KUKA KRL program: fahrwege_big.src

&ACCESS RVO1
&REL 803
&COMMENT Rack 1 Place
&PARAM DISKPATH = KRC:\R1\Program\Unterprogramme
DEF  fahrwege_big( )
  ;FOLD INI;%{PE}
  ;FOLD BASISTECH INI
  GLOBAL INTERRUPT DECL 3 WHEN $STOPMESS==TRUE DO IR_STOPM ( )
  INTERRUPT ON 3
  BAS (#INITMOV,0 )
  ;ENDFOLD (BASISTECH INI)
  ;FOLD USER INI
  ;Make your modifications here

  ;ENDFOLD (USER INI)
  ;ENDFOLD (INI)

;***************************************************
; SAK herstellen
PTP $POS_ACT
;***************************************************

;---------------------------------
; Roboter in Grundstellung fahren
;---------------------------------
IF NOT ($IN_HOME OR $IN_HOME1 OR $IN_HOME2 OR $IN_HOME3) THEN
  UP_Rueckzug( )
ENDIF

;***************************************************
;      Unterprogramme fuer Produktionsbetrieb
;***************************************************

;***************************************************
; Satzanwahl auf gewuenschtes Unterprogramm
LOOP
  WAIT SEC 0.1
ENDLOOP
;***************************************************

HALT
UP_Place_R1_L1_S1( )
HALT
UP_Place_R1_L1_S2( )
HALT
UP_Place_R1_L1_S3( )
HALT
UP_Place_R1_L1_S4( )
HALT
UP_Place_R1_L2_S1( )
HALT
UP_Place_R1_L2_S2( )
HALT
UP_Place_R1_L2_S3( )
HALT
UP_Place_R1_L2_S4( )
HALT
UP_Place_R1_L3_S1( )
HALT
UP_Place_R1_L3_S2( )
HALT
UP_Place_R1_L3_S3( )
HALT
UP_Place_R1_L3_S4( )
HALT
UP_Place_R1_L4_S1( )
HALT
UP_Place_R1_L4_S2( )
HALT
UP_Place_R1_L4_S3( )
HALT
UP_Place_R1_L4_S4( )
HALT
UP_Place_R1_L5_S1( )
HALT
UP_Place_R1_L5_S2( )
HALT
UP_Place_R1_L5_S3( )
HALT
UP_Place_R1_L5_S4( )
HALT
UP_Place_R1_L6_S1( )
HALT
UP_Place_R1_L6_S2( )
HALT
UP_Place_R1_L6_S3( )
HALT
UP_Place_R1_L6_S4( )
HALT
UP_Place_R1_L7_S1( )
HALT
UP_Place_R1_L7_S2( )
HALT
UP_Place_R1_L7_S3( )
HALT
UP_Place_R1_L7_S4( )
HALT
UP_Place_R1_L8_S1( )
HALT
UP_Place_R1_L8_S2( )
HALT
UP_Place_R1_L8_S3( )
HALT
UP_Place_R1_L8_S4( )
HALT
UP_Rueckzug_R1Place( )
HALT
;***************************************************

END

; ##################################################

GLOBAL DEF UP_Place_R1_L1_S1( )
;***************************************************
; Place part on:
;    Rack  1
;    Level 1
;    Shelf 1
;***************************************************
;FOLD Preconditions - Vorraussetzungen
;***************************************************
; Enable collision detection
;FOLD COLLDETECT SetLimits Axis1: 150 % Axis2: 200 % Axis3: 150 % Axis4: 200 % Axis5: 150 % Axis6: 150 % ;%{PE}
;FOLD Parameters ;%{h}
;Params IlfProvider=kukaroboter.basistech.inlineforms.colldetect.setlimits; CollDetect.Command=SetLimits; CollDetect.Axis1=150; CollDetect.Axis2=200; CollDetect.Axis3=150; CollDetect.Axis4=200; CollDetect.Axis5=150; CollDetect.Axis6=150
;ENDFOLD
SET_TQ_VALUES(150, 200, 150, 200, 150, 150)
;ENDFOLD
;***************************************************
; Check for part in gripper (tool 2).
CheckPartPresent(OCCUPIED_GRIPPER,PART_ON_TOOL_2)
;***************************************************
; Enable part lost detection for tool 2
SetPartLostDetection(PART_ON_TOOL_2)
;***************************************************
; Set load data.
SetLoadData( )
;***************************************************
; Robot has to start from home position.
IF NOT $IN_HOME1 THEN
  UP_HomeToHome(1)
ENDIF
;***************************************************
;ENDFOLD

TRIGGER WHEN DISTANCE=1 DELAY=-1 DO Schrittmerker_R1Place(10002,10002,FHOME1,$nullframe,XHOME1) PRIO=-1
;FOLD PTP HOME1 Vel=12 % PHome1;%{PE}%R8.3.21,%MKUKATPBASIS,%CMOVE,%VPTP,%P 1:PTP, 2:HOME1, 3:, 5:12, 7:PHome1
$BWDSTART=FALSE
PDAT_ACT= PPHome1
FDAT_ACT= FHOME1
BAS(#PTP_PARAMS,12)
PTP XHOME1
;ENDFOLD

;***************************************************
;FOLD Area clearence handshake.
IF NOT $FLAG[M_Inbetriebnahme] THEN
  ;-------------------------------------------------
  ; Request area clearence.
  AnfStoer_Store1_1_A99=SET_REQUEST
  ;-------------------------------------------------
  ; Wait for area clearence from PLC.
  WAIT_FOR_INPUT("Frg_Storage1_1_E67",TRUE)
  ;-------------------------------------------------
  ; Reset area clearence request.
  AnfStoer_Store1_1_A99=RESET_REQUEST
  ;-------------------------------------------------
  ; start cyclic clearence check
  $CYCFLAG[ciFreigabeSPS]=Frg_Storage1_1_E67
  ;-------------------------------------------------
ENDIF
;***************************************************
; set "robot in area"
RobAusStorage1_1_A67=SET_IN_AREA
;ENDFOLD
;***************************************************

;***************************************************
;FOLD Check for Teachmode
IF $FLAG[M_Teachen] THEN
  WAIT FOR $T1
ENDIF
;ENDFOLD
;***************************************************

; move to the rack
TRIGGER WHEN DISTANCE=1 DELAY=-1 DO Schrittmerker_R1Place(10003,10002,FPlace_R1_L1_S1_VP1,XPlace_R1_L1_S1_VP1) PRIO=-1
;FOLD PTP Place_R1_L1_S1_VP1 CONT Vel=12 % PPlace_R1_L1_S1_VP1 Tool[2]:Lower Gripper Base[0];%{PE}%R8.3.21,%MKUKATPBASIS,%CMOVE,%VPTP,%P 1:PTP, 2:Place_R1_L1_S1_VP1, 3:C_DIS, 5:12, 7:PPlace_R1_L1_S1_VP1
$BWDSTART=FALSE
PDAT_ACT= PPPlace_R1_L1_S1_VP1
FDAT_ACT= FPlace_R1_L1_S1_VP1
BAS(#PTP_PARAMS,12)
PTP XPlace_R1_L1_S1_VP1 C_DIS
;ENDFOLD
TRIGGER WHEN DISTANCE=1 DELAY=-1 DO Schrittmerker_R1Place(10004,10003,FPlace_R1_L1_S1_VP2,XPlace_R1_L1_S1_VP2) PRIO=-1
;FOLD PTP Place_R1_L1_S1_VP2 CONT Vel=12 % PPlace_R1_L1_S1_VP2 Tool[2]:Lower Gripper Base[0];%{PE}%R8.3.21,%MKUKATPBASIS,%CMOVE,%VPTP,%P 1:PTP, 2:Place_R1_L1_S1_VP2, 3:C_DIS, 5:12, 7:PPlace_R1_L1_S1_VP2
$BWDSTART=FALSE
PDAT_ACT= PPPlace_R1_L1_S1_VP2
FDAT_ACT= FPlace_R1_L1_S1_VP2
BAS(#PTP_PARAMS,12)
PTP XPlace_R1_L1_S1_VP2 C_DIS
;ENDFOLD
TRIGGER WHEN DISTANCE=1 DELAY=-1 DO Schrittmerker_R1Place(10005,10004,FPlace_R1_L1_S1_VP3,XPlace_R1_L1_S1_VP3) PRIO=-1
;FOLD PTP Place_R1_L1_S1_VP3 CONT Vel=12 % PPlace_R1_L1_S1_VP3 Tool[2]:Lower Gripper Base[0];%{PE}%R8.3.21,%MKUKATPBASIS,%CMOVE,%VPTP,%P 1:PTP, 2:Place_R1_L1_S1_VP3, 3:C_DIS, 5:12, 7:PPlace_R1_L1_S1_VP3
$BWDSTART=FALSE
PDAT_ACT= PPPlace_R1_L1_S1_VP3
FDAT_ACT= FPlace_R1_L1_S1_VP3
BAS(#PTP_PARAMS,12)
PTP XPlace_R1_L1_S1_VP3 C_DIS
;ENDFOLD
TRIGGER WHEN DISTANCE=1 DELAY=-1 DO Schrittmerker_R1Place(10006,10005,FPlace_R1_L1_S1_VP4,XPlace_R1_L1_S1_VP4) PRIO=-1
;FOLD PTP Place_R1_L1_S1_VP4 CONT Vel=12 % PPlace_R1_L1_S1_VP4 Tool[2]:Lower Gripper Base[0];%{PE}%R8.3.21,%MKUKATPBASIS,%CMOVE,%VPTP,%P 1:PTP, 2:Place_R1_L1_S1_VP4, 3:C_DIS, 5:12, 7:PPlace_R1_L1_S1_VP4
$BWDSTART=FALSE
PDAT_ACT= PPPlace_R1_L1_S1_VP4
FDAT_ACT= FPlace_R1_L1_S1_VP4
BAS(#PTP_PARAMS,12)
PTP XPlace_R1_L1_S1_VP4 C_DIS
;ENDFOLD
TRIGGER WHEN DISTANCE=1 DELAY=-1 DO Schrittmerker_R1Place(10007,10006,FPlace_R1_L1_S1_VP5,XPlace_R1_L1_S1_VP5) PRIO=-1
;FOLD PTP Place_R1_L1_S1_VP5 CONT Vel=12 % PPlace_R1_L1_S1_VP5 Tool[2]:Lower Gripper Base[0];%{PE}%R8.3.21,%MKUKATPBASIS,%CMOVE,%VPTP,%P 1:PTP, 2:Place_R1_L1_S1_VP5, 3:C_DIS, 5:12, 7:PPlace_R1_L1_S1_VP5
$BWDSTART=FALSE
PDAT_ACT= PPPlace_R1_L1_S1_VP5
FDAT_ACT= FPlace_R1_L1_S1_VP5
BAS(#PTP_PARAMS,12)
PTP XPlace_R1_L1_S1_VP5 C_DIS
;ENDFOLD
TRIGGER WHEN DISTANCE=1 DELAY=-1 DO Schrittmerker_R1Place(10008,10007,FPlace_R1_L1_S1_VP6,XPlace_R1_L1_S1_VP6) PRIO=-1
;FOLD PTP Place_R1_L1_S1_VP6 CONT Vel=12 % PPlace_R1_L1_S1_VP6 Tool[2]:Lower Gripper Base[1]:Rack1;%{PE}%R8.3.21,%MKUKATPBASIS,%CMOVE,%VPTP,%P 1:PTP, 2:Place_R1_L1_S1_VP6, 3:C_DIS, 5:12, 7:PPlace_R1_L1_S1_VP6
$BWDSTART=FALSE
PDAT_ACT= PPPlace_R1_L1_S1_VP6
FDAT_ACT= FPlace_R1_L1_S1_VP6
BAS(#PTP_PARAMS,12)
PTP XPlace_R1_L1_S1_VP6 C_DIS
;ENDFOLD

TRIGGER WHEN DISTANCE=1 DELAY=-1 DO Schrittmerker_R1Place(10009,10008,FPlace_R1_L1_S1_Check,XPlace_R1_L1_S1_Check) PRIO=-1
;FOLD PTP Place_R1_L1_S1_Check Vel=12 % PPlace_R1_L1_S1_Check Tool[2]:Lower Gripper Base[1]:Rack1;%{PE}%R8.3.21,%MKUKATPBASIS,%CMOVE,%VPTP,%P 1:PTP, 2:Place_R1_L1_S1_Check, 3:, 5:12, 7:PPlace_R1_L1_S1_Check
$BWDSTART=FALSE
PDAT_ACT= PPPlace_R1_L1_S1_Check
FDAT_ACT= FPlace_R1_L1_S1_Check
BAS(#PTP_PARAMS,12)
PTP XPlace_R1_L1_S1_Check
;ENDFOLD

;***************************************************
;FOLD Pruefe Platz frei
IF (DetectPart(CHECK_SHELF,PLACE)==OCCUPIED) THEN
  UP_Rueckzug_R1Place( )
  RETURN
ENDIF
;ENDFOLD
;***************************************************

TRIGGER WHEN DISTANCE=1 DELAY=-1 DO Schrittmerker_R1Place(10010,10009,FPlace_R1_L1_S1_VP7,XPlace_R1_L1_S1_VP7) PRIO=-1
;FOLD LIN Place_R1_L1_S1_VP7 CONT Vel=0.5 m/s LPlace_R1_L1_S1_VP7 Tool[2]:Lower Gripper Base[1]:Rack1;%{PE}%R8.3.21,%MKUKATPBASIS,%CMOVE,%VLIN,%P 1:LIN, 2:Place_R1_L1_S1_VP7, 3:C_DIS C_DIS, 5:0.5, 7:LPlace_R1_L1_S1_VP7
$BWDSTART=FALSE
LDAT_ACT= LLPlace_R1_L1_S1_VP7
FDAT_ACT= FPlace_R1_L1_S1_VP7
BAS(#CP_PARAMS,0.5)
LIN XPlace_R1_L1_S1_VP7 C_DIS C_DIS
;ENDFOLD
TRIGGER WHEN DISTANCE=1 DELAY=-1 DO Schrittmerker_R1Place(10011,10010,FPlace_R1_L1_S1_VP8,XPlace_R1_L1_S1_VP8) PRIO=-1
;FOLD LIN Place_R1_L1_S1_VP8 CONT Vel=0.5 m/s LPlace_R1_L1_S1_VP8 Tool[2]:Lower Gripper Base[1]:Rack1;%{PE}%R8.3.21,%MKUKATPBASIS,%CMOVE,%VLIN,%P 1:LIN, 2:Place_R1_L1_S1_VP8, 3:C_DIS C_DIS, 5:0.5, 7:LPlace_R1_L1_S1_VP8
$BWDSTART=FALSE
LDAT_ACT= LLPlace_R1_L1_S1_VP8
FDAT_ACT= FPlace_R1_L1_S1_VP8
BAS(#CP_PARAMS,0.5)
LIN XPlace_R1_L1_S1_VP8 C_DIS C_DIS
;ENDFOLD
TRIGGER WHEN DISTANCE=1 DELAY=-1 DO Schrittmerker_R1Place(10012,10011,FPlace_R1_L1_S1_VP9,XPlace_R1_L1_S1_VP9) PRIO=-1
;FOLD LIN Place_R1_L1_S1_VP9 CONT Vel=0.5 m/s LPlace_R1_L1_S1_VP9 Tool[2]:Lower Gripper Base[1]:Rack1;%{PE}%R8.3.21,%MKUKATPBASIS,%CMOVE,%VLIN,%P 1:LIN, 2:Place_R1_L1_S1_VP9, 3:C_DIS C_DIS, 5:0.5, 7:LPlace_R1_L1_S1_VP9
$BWDSTART=FALSE
LDAT_ACT= LLPlace_R1_L1_S1_VP9
FDAT_ACT= FPlace_R1_L1_S1_VP9
BAS(#CP_PARAMS,0.5)
LIN XPlace_R1_L1_S1_VP9 C_DIS C_DIS
;ENDFOLD

;FOLD Test the way back home - part 1
CONTINUE
IF ($FLAG[M_Test_GrdstFahren1] AND NOT $FLAG[M_Test_GrdstFahren2]) THEN
  $FLAG[M_Test_GrdstFahren2]=TRUE
  UP_Rueckzug( )
  RETURN
ENDIF
;ENDFOLD

;-------------------------------
; Place part position
;-------------------------------
TRIGGER WHEN DISTANCE=1 DELAY=-1 DO Schrittmerker_R1Place(10013,10014,FPlace_R1_L1_S1_AP,XPlace_R1_L1_S1_AP) PRIO=-1
;FOLD LIN Place_R1_L1_S1_AP Vel=0.2 m/s LPlace_R1_L1_S1_AP Tool[2]:Lower Gripper Base[1]:Rack1;%{PE}%R8.3.21,%MKUKATPBASIS,%CMOVE,%VLIN,%P 1:LIN, 2:Place_R1_L1_S1_AP, 3:, 5:0.2, 7:LPlace_R1_L1_S1_AP
$BWDSTART=FALSE
LDAT_ACT= LLPlace_R1_L1_S1_AP
FDAT_ACT= FPlace_R1_L1_S1_AP
BAS(#CP_PARAMS,0.2)
LIN XPlace_R1_L1_S1_AP
;ENDFOLD

;FOLD Test the way back home - part 2
CONTINUE
IF $FLAG[M_Test_GrdstFahren2] THEN
  $FLAG[M_Test_GrdstFahren2]=FALSE
  UP_Rueckzug( )
  RETURN
ENDIF
;ENDFOLD

;***************************************************
; Disable part lost detection
SetPartLostDetection(NO_PART)
;***************************************************

TRIGGER WHEN DISTANCE=1 DELAY=-1 DO Schrittmerker_R1Place(10014,10015,FPlace_R1_L1_S1_NP1,XPlace_R1_L1_S1_NP1) PRIO=-1
;FOLD LIN Place_R1_L1_S1_NP1 Vel=0.2 m/s LPlace_R1_L1_S1_NP1 Tool[2]:Lower Gripper Base[1]:Rack 1 ;%{PE}
;FOLD Parameters ;%{h}
;Params IlfProvider=kukaroboter.basistech.inlineforms.movement.old; Kuka.IsGlobalPoint=False; Kuka.PointName=Place_R1_L1_S1_NP1; Kuka.BlendingEnabled=False; Kuka.MoveDataName=LPlace_R1_L1_S1_NP1; Kuka.VelocityPath=0.2; Kuka.CurrentCDSetIndex=0; Kuka.MovementParameterFieldEnabled=True; IlfCommand=LIN
;ENDFOLD
$BWDSTART = FALSE
LDAT_ACT = LLPlace_R1_L1_S1_NP1
FDAT_ACT = FPlace_R1_L1_S1_NP1
BAS(#CP_PARAMS, 0.2)
SET_CD_PARAMS (0)
LIN XPlace_R1_L1_S1_NP1
;ENDFOLD

;***************************************************
; Check for part present (empty gripper)
CheckPartPresent(EMPTY_GRIPPER)
;***************************************************
; set load data
SetLoadData( )
;***************************************************

TRIGGER WHEN DISTANCE=1 DELAY=-1 DO Schrittmerker_R1Place(10015,10016,FPlace_R1_L1_S1_NP2,XPlace_R1_L1_S1_NP2) PRIO=-1
;FOLD LIN Place_R1_L1_S1_NP2 CONT Vel=0.5 m/s LPlace_R1_L1_S1_NP2 Tool[2]:Lower Gripper Base[1]:Rack1;%{PE}%R8.3.21,%MKUKATPBASIS,%CMOVE,%VLIN,%P 1:LIN, 2:Place_R1_L1_S1_NP2, 3:C_DIS C_DIS, 5:0.5, 7:LPlace_R1_L1_S1_NP2
$BWDSTART=FALSE
LDAT_ACT= LLPlace_R1_L1_S1_NP2
FDAT_ACT= FPlace_R1_L1_S1_NP2
BAS(#CP_PARAMS,0.5)
LIN XPlace_R1_L1_S1_NP2 C_DIS C_DIS
;ENDFOLD
TRIGGER WHEN DISTANCE=1 DELAY=-1 DO Schrittmerker_R1Place(10016,10017,FPlace_R1_L1_S1_NP3,XPlace_R1_L1_S1_NP3) PRIO=-1
;FOLD LIN Place_R1_L1_S1_NP3 Vel=0.5 m/s LPlace_R1_L1_S1_NP3 Tool[2]:Lower Gripper Base[1]:Rack1;%{PE}%R8.3.21,%MKUKATPBASIS,%CMOVE,%VLIN,%P 1:LIN, 2:Place_R1_L1_S1_NP3, 3:, 5:0.5, 7:LPlace_R1_L1_S1_NP3
$BWDSTART=FALSE
LDAT_ACT= LLPlace_R1_L1_S1_NP3
FDAT_ACT= FPlace_R1_L1_S1_NP3
BAS(#CP_PARAMS,0.5)
LIN XPlace_R1_L1_S1_NP3
;ENDFOLD
TRIGGER WHEN DISTANCE=1 DELAY=-1 DO Schrittmerker_R1Place(10017,10018,FPlace_R1_L1_S1_NP4,XPlace_R1_L1_S1_NP4) PRIO=-1
;FOLD PTP Place_R1_L1_S1_NP4 CONT Vel=100 % PPlace_R1_L1_S1_NP4 Tool[2]:Lower Gripper Base[1]:Rack1;%{PE}%R8.3.21,%MKUKATPBASIS,%CMOVE,%VPTP,%P 1:PTP, 2:Place_R1_L1_S1_NP4, 3:C_DIS, 5:100, 7:PPlace_R1_L1_S1_NP4
$BWDSTART=FALSE
PDAT_ACT= PPPlace_R1_L1_S1_NP4
FDAT_ACT= FPlace_R1_L1_S1_NP4
BAS(#PTP_PARAMS,100)
PTP XPlace_R1_L1_S1_NP4 C_DIS
;ENDFOLD
TRIGGER WHEN DISTANCE=1 DELAY=-1 DO Schrittmerker_R1Place(10018,10019,FPlace_R1_L1_S1_NP5,XPlace_R1_L1_S1_NP5) PRIO=-1
;FOLD PTP Place_R1_L1_S1_NP5 CONT Vel=100 % PPlace_R1_L1_S1_NP5 Tool[2]:Lower Gripper Base[0];%{PE}%R8.3.21,%MKUKATPBASIS,%CMOVE,%VPTP,%P 1:PTP, 2:Place_R1_L1_S1_NP5, 3:C_DIS, 5:100, 7:PPlace_R1_L1_S1_NP5
$BWDSTART=FALSE
PDAT_ACT= PPPlace_R1_L1_S1_NP5
FDAT_ACT= FPlace_R1_L1_S1_NP5
BAS(#PTP_PARAMS,100)
PTP XPlace_R1_L1_S1_NP5 C_DIS
;ENDFOLD
TRIGGER WHEN DISTANCE=1 DELAY=-1 DO Schrittmerker_R1Place(10019,10020,FPlace_R1_L1_S1_NP6,XPlace_R1_L1_S1_NP6) PRIO=-1
;FOLD PTP Place_R1_L1_S1_NP6 CONT Vel=100 % PPlace_R1_L1_S1_NP6 Tool[2]:Lower Gripper Base[0];%{PE}%R8.3.21,%MKUKATPBASIS,%CMOVE,%VPTP,%P 1:PTP, 2:Place_R1_L1_S1_NP6, 3:C_DIS, 5:100, 7:PPlace_R1_L1_S1_NP6
$BWDSTART=FALSE
PDAT_ACT= PPPlace_R1_L1_S1_NP6
FDAT_ACT= FPlace_R1_L1_S1_NP6
BAS(#PTP_PARAMS,100)
PTP XPlace_R1_L1_S1_NP6 C_DIS
;ENDFOLD
TRIGGER WHEN DISTANCE=1 DELAY=-1 DO Schrittmerker_R1Place(10020,10021,FPlace_R1_L1_S1_NP7,XPlace_R1_L1_S1_NP7) PRIO=-1
;FOLD PTP Place_R1_L1_S1_NP7 CONT Vel=100 % PPlace_R1_L1_S1_NP7 Tool[2]:Lower Gripper Base[0];%{PE}%R8.3.21,%MKUKATPBASIS,%CMOVE,%VPTP,%P 1:PTP, 2:Place_R1_L1_S1_NP7, 3:C_DIS, 5:100, 7:PPlace_R1_L1_S1_NP7
$BWDSTART=FALSE
PDAT_ACT= PPPlace_R1_L1_S1_NP7
FDAT_ACT= FPlace_R1_L1_S1_NP7
BAS(#PTP_PARAMS,100)
PTP XPlace_R1_L1_S1_NP7 C_DIS
;ENDFOLD
TRIGGER WHEN DISTANCE=1 DELAY=-1 DO Schrittmerker_R1Place(10021,10022,FPlace_R1_L1_S1_NP8,XPlace_R1_L1_S1_NP8) PRIO=-1
;FOLD PTP Place_R1_L1_S1_NP8 CONT Vel=100 % PPlace_R1_L1_S1_NP8 Tool[2]:Lower Gripper Base[0];%{PE}%R8.3.21,%MKUKATPBASIS,%CMOVE,%VPTP,%P 1:PTP, 2:Place_R1_L1_S1_NP8, 3:C_DIS, 5:100, 7:PPlace_R1_L1_S1_NP8
$BWDSTART=FALSE
PDAT_ACT= PPPlace_R1_L1_S1_NP8
FDAT_ACT= FPlace_R1_L1_S1_NP8
BAS(#PTP_PARAMS,100)
PTP XPlace_R1_L1_S1_NP8 C_DIS
;ENDFOLD
TRIGGER WHEN DISTANCE=1 DELAY=-1 DO Schrittmerker_R1Place(10022,10023,FPlace_R1_L1_S1_NP9,XPlace_R1_L1_S1_NP9) PRIO=-1
;FOLD PTP Place_R1_L1_S1_NP9 CONT Vel=100 % PPlace_R1_L1_S1_NP9 Tool[2]:Lower Gripper Base[0];%{PE}%R8.3.21,%MKUKATPBASIS,%CMOVE,%VPTP,%P 1:PTP, 2:Place_R1_L1_S1_NP9, 3:C_DIS, 5:100, 7:PPlace_R1_L1_S1_NP9
$BWDSTART=FALSE
PDAT_ACT= PPPlace_R1_L1_S1_NP9
FDAT_ACT= FPlace_R1_L1_S1_NP9
BAS(#PTP_PARAMS,100)
PTP XPlace_R1_L1_S1_NP9 C_DIS
;ENDFOLD

TRIGGER WHEN DISTANCE=1 DELAY=-1 DO Schrittmerker_R1Place(10023,10002,FHOME1,$nullframe,XHOME1) PRIO=-1
;FOLD PTP HOME1 Vel=100 % PHome1;%{PE}%R8.3.21,%MKUKATPBASIS,%CMOVE,%VPTP,%P 1:PTP, 2:HOME1, 3:, 5:100, 7:PHome1
$BWDSTART=FALSE
PDAT_ACT= PPHome1
FDAT_ACT= FHOME1
BAS(#PTP_PARAMS,100)
PTP XHOME1
;ENDFOLD

;***************************************************
;FOLD Final tasks.
; Robot out of area Rack 1 Level 1
RobAusStorage1_1_A67=RESET_IN_AREA
;***************************************************
; stop cyclic clearence check
$CYCFLAG[ciFreigabeSPS]=DISABLE_MONITORING
;***************************************************
; Disable collision detection
;FOLD COLLDETECT Off ;%{PE}
;FOLD Parameters ;%{h}
;Params IlfProvider=kukaroboter.basistech.inlineforms.colldetect.off; CollDetect.Command=Off
;ENDFOLD
USE_CD_PARAMS(0)
;ENDFOLD
;***************************************************
;ENDFOLD
;***************************************************

END

; ##################################################

GLOBAL DEF UP_Place_R1_L1_S2( )
;***************************************************
; Place part on:
;    Rack  1
;    Level 1
;    Shelf 2
;***************************************************
;FOLD Preconditions - Vorraussetzungen
;***************************************************
; Enable collision detection
;FOLD COLLDETECT SetLimits Axis1: 150 % Axis2: 200 % Axis3: 150 % Axis4: 200 % Axis5: 150 % Axis6: 150 % ;%{PE}
;FOLD Parameters ;%{h}
;Params IlfProvider=kukaroboter.basistech.inlineforms.colldetect.setlimits; CollDetect.Command=SetLimits; CollDetect.Axis1=150; CollDetect.Axis2=200; CollDetect.Axis3=150; CollDetect.Axis4=200; CollDetect.Axis5=150; CollDetect.Axis6=150
;ENDFOLD
SET_TQ_VALUES(150, 200, 150, 200, 150, 150)
;ENDFOLD
;***************************************************
; Check for part in gripper (tool 2).
CheckPartPresent(OCCUPIED_GRIPPER,PART_ON_TOOL_2)
;***************************************************
; Enable part lost detection for tool 2
SetPartLostDetection(PART_ON_TOOL_2)
;***************************************************
; Set load data.
SetLoadData( )
;***************************************************
; Robot has to start from home position.
IF NOT $IN_HOME1 THEN
  UP_HomeToHome(1)
ENDIF
;***************************************************
;ENDFOLD

TRIGGER WHEN DISTANCE=1 DELAY=-1 DO Schrittmerker_R1Place(10002,10002,FHOME1,$nullframe,XHOME1) PRIO=-1
;FOLD PTP HOME1 Vel=12 % PHome1;%{PE}%R8.3.21,%MKUKATPBASIS,%CMOVE,%VPTP,%P 1:PTP, 2:HOME1, 3:, 5:12, 7:PHome1
$BWDSTART=FALSE
PDAT_ACT= PPHome1
FDAT_ACT= FHOME1
BAS(#PTP_PARAMS,12)
PTP XHOME1
;ENDFOLD

;***************************************************
;FOLD Area clearence handshake.
IF NOT $FLAG[M_Inbetriebnahme] THEN
  ;-------------------------------------------------
  ; Request area clearence.
  AnfStoer_Store1_1_A99=SET_REQUEST
  ;-------------------------------------------------
  ; Wait for area clearence from PLC.
  WAIT_FOR_INPUT("Frg_Storage1_1_E67",TRUE)
  ;-------------------------------------------------
  ; Reset area clearence request.
  AnfStoer_Store1_1_A99=RESET_REQUEST
  ;-------------------------------------------------
  ; start cyclic clearence check
  $CYCFLAG[ciFreigabeSPS]=Frg_Storage1_1_E67
  ;-------------------------------------------------
ENDIF
;***************************************************
; set "robot in area"
RobAusStorage1_1_A67=SET_IN_AREA
;ENDFOLD
;***************************************************

;***************************************************
;FOLD Check for Teachmode
IF $FLAG[M_Teachen] THEN
  WAIT FOR $T1
ENDIF
;ENDFOLD
;***************************************************

; move to the rack
TRIGGER WHEN DISTANCE=1 DELAY=-1 DO Schrittmerker_R1Place(10025,10002,FPlace_R1_L1_S2_VP1,XPlace_R1_L1_S2_VP1) PRIO=-1
;FOLD PTP Place_R1_L1_S2_VP1 CONT Vel=12 % PPlace_R1_L1_S2_VP1 Tool[2]:Lower Gripper Base[0];%{PE}%R8.3.21,%MKUKATPBASIS,%CMOVE,%VPTP,%P 1:PTP, 2:Place_R1_L1_S2_VP1, 3:C_DIS, 5:12, 7:PPlace_R1_L1_S2_VP1
$BWDSTART=FALSE
PDAT_ACT= PPPlace_R1_L1_S2_VP1
FDAT_ACT= FPlace_R1_L1_S2_VP1
BAS(#PTP_PARAMS,12)
PTP XPlace_R1_L1_S2_VP1 C_DIS
;ENDFOLD
TRIGGER WHEN DISTANCE=1 DELAY=-1 DO Schrittmerker_R1Place(10026,10025,FPlace_R1_L1_S2_VP2,XPlace_R1_L1_S2_VP2) PRIO=-1
;FOLD PTP Place_R1_L1_S2_VP2 CONT Vel=12 % PPlace_R1_L1_S2_VP2 Tool[2]:Lower Gripper Base[0];%{PE}%R8.3.21,%MKUKATPBASIS,%CMOVE,%VPTP,%P 1:PTP, 2:Place_R1_L1_S2_VP2, 3:C_DIS, 5:12, 7:PPlace_R1_L1_S2_VP2
$BWDSTART=FALSE
PDAT_ACT= PPPlace_R1_L1_S2_VP2
FDAT_ACT= FPlace_R1_L1_S2_VP2
BAS(#PTP_PARAMS,12)
PTP XPlace_R1_L1_S2_VP2 C_DIS
;ENDFOLD
TRIGGER WHEN DISTANCE=1 DELAY=-1 DO Schrittmerker_R1Place(10027,10026,FPlace_R1_L1_S2_VP3,XPlace_R1_L1_S2_VP3) PRIO=-1
;FOLD PTP Place_R1_L1_S2_VP3 CONT Vel=12 % PPlace_R1_L1_S2_VP3 Tool[2]:Lower Gripper Base[0];%{PE}%R8.3.21,%MKUKATPBASIS,%CMOVE,%VPTP,%P 1:PTP, 2:Place_R1_L1_S2_VP3, 3:C_DIS, 5:12, 7:PPlace_R1_L1_S2_VP3
$BWDSTART=FALSE
PDAT_ACT= PPPlace_R1_L1_S2_VP3
FDAT_ACT= FPlace_R1_L1_S2_VP3
BAS(#PTP_PARAMS,12)
PTP XPlace_R1_L1_S2_VP3 C_DIS
;ENDFOLD
TRIGGER WHEN DISTANCE=1 DELAY=-1 DO Schrittmerker_R1Place(10028,10027,FPlace_R1_L1_S2_VP4,XPlace_R1_L1_S2_VP4) PRIO=-1
;FOLD PTP Place_R1_L1_S2_VP4 CONT Vel=12 % PPlace_R1_L1_S2_VP4 Tool[2]:Lower Gripper Base[0];%{PE}%R8.3.21,%MKUKATPBASIS,%CMOVE,%VPTP,%P 1:PTP, 2:Place_R1_L1_S2_VP4, 3:C_DIS, 5:12, 7:PPlace_R1_L1_S2_VP4
$BWDSTART=FALSE
PDAT_ACT= PPPlace_R1_L1_S2_VP4
FDAT_ACT= FPlace_R1_L1_S2_VP4
BAS(#PTP_PARAMS,12)
PTP XPlace_R1_L1_S2_VP4 C_DIS
;ENDFOLD
TRIGGER WHEN DISTANCE=1 DELAY=-1 DO Schrittmerker_R1Place(10029,10028,FPlace_R1_L1_S2_VP5,XPlace_R1_L1_S2_VP5) PRIO=-1
;FOLD PTP Place_R1_L1_S2_VP5 CONT Vel=12 % PPlace_R1_L1_S2_VP5 Tool[2]:Lower Gripper Base[0];%{PE}%R8.3.21,%MKUKATPBASIS,%CMOVE,%VPTP,%P 1:PTP, 2:Place_R1_L1_S2_VP5, 3:C_DIS, 5:12, 7:PPlace_R1_L1_S2_VP5
$BWDSTART=FALSE
PDAT_ACT= PPPlace_R1_L1_S2_VP5
FDAT_ACT= FPlace_R1_L1_S2_VP5
BAS(#PTP_PARAMS,12)
PTP XPlace_R1_L1_S2_VP5 C_DIS
;ENDFOLD
TRIGGER WHEN DISTANCE=1 DELAY=-1 DO Schrittmerker_R1Place(10030,10029,FPlace_R1_L1_S2_VP6,XPlace_R1_L1_S2_VP6) PRIO=-1
;FOLD PTP Place_R1_L1_S2_VP6 CONT Vel=12 % PPlace_R1_L1_S2_VP6 Tool[2]:Lower Gripper Base[1]:Rack1;%{PE}%R8.3.21,%MKUKATPBASIS,%CMOVE,%VPTP,%P 1:PTP, 2:Place_R1_L1_S2_VP6, 3:C_DIS, 5:12, 7:PPlace_R1_L1_S2_VP6
$BWDSTART=FALSE
PDAT_ACT= PPPlace_R1_L1_S2_VP6
FDAT_ACT= FPlace_R1_L1_S2_VP6
BAS(#PTP_PARAMS,12)
PTP XPlace_R1_L1_S2_VP6 C_DIS
;ENDFOLD

TRIGGER WHEN DISTANCE=1 DELAY=-1 DO Schrittmerker_R1Place(10031,10030,FPlace_R1_L1_S2_Check,XPlace_R1_L1_S2_Check) PRIO=-1
;FOLD PTP Place_R1_L1_S2_Check Vel=12 % PPlace_R1_L1_S2_Check Tool[2]:Lower Gripper Base[1]:Rack1;%{PE}%R8.3.21,%MKUKATPBASIS,%CMOVE,%VPTP,%P 1:PTP, 2:Place_R1_L1_S2_Check, 3:, 5:12, 7:PPlace_R1_L1_S2_Check
$BWDSTART=FALSE
PDAT_ACT= PPPlace_R1_L1_S2_Check
FDAT_ACT= FPlace_R1_L1_S2_Check
BAS(#PTP_PARAMS,12)
PTP XPlace_R1_L1_S2_Check
;ENDFOLD

;***************************************************
;FOLD Pruefe Platz frei
IF (DetectPart(CHECK_SHELF,PLACE)==OCCUPIED) THEN
  UP_Rueckzug_R1Place( )
  RETURN
ENDIF
;ENDFOLD
;***************************************************

TRIGGER WHEN DISTANCE=1 DELAY=-1 DO Schrittmerker_R1Place(10032,10031,FPlace_R1_L1_S2_VP7,XPlace_R1_L1_S2_VP7) PRIO=-1
;FOLD LIN Place_R1_L1_S2_VP7 CONT Vel=0.5 m/s LPlace_R1_L1_S2_VP7 Tool[2]:Lower Gripper Base[1]:Rack1;%{PE}%R8.3.21,%MKUKATPBASIS,%CMOVE,%VLIN,%P 1:LIN, 2:Place_R1_L1_S2_VP7, 3:C_DIS C_DIS, 5:0.5, 7:LPlace_R1_L1_S2_VP7
$BWDSTART=FALSE
LDAT_ACT= LLPlace_R1_L1_S2_VP7
FDAT_ACT= FPlace_R1_L1_S2_VP7
BAS(#CP_PARAMS,0.5)
LIN XPlace_R1_L1_S2_VP7 C_DIS C_DIS
;ENDFOLD
TRIGGER WHEN DISTANCE=1 DELAY=-1 DO Schrittmerker_R1Place(10033,10032,FPlace_R1_L1_S2_VP8,XPlace_R1_L1_S2_VP8) PRIO=-1
;FOLD LIN Place_R1_L1_S2_VP8 CONT Vel=0.5 m/s LPlace_R1_L1_S2_VP8 Tool[2]:Lower Gripper Base[1]:Rack1;%{PE}%R8.3.21,%MKUKATPBASIS,%CMOVE,%VLIN,%P 1:LIN, 2:Place_R1_L1_S2_VP8, 3:C_DIS C_DIS, 5:0.5, 7:LPlace_R1_L1_S2_VP8
$BWDSTART=FALSE
LDAT_ACT= LLPlace_R1_L1_S2_VP8
FDAT_ACT= FPlace_R1_L1_S2_VP8
BAS(#CP_PARAMS,0.5)
LIN XPlace_R1_L1_S2_VP8 C_DIS C_DIS
;ENDFOLD

;FOLD Test the way back home - part 1
CONTINUE
IF ($FLAG[M_Test_GrdstFahren1] AND NOT $FLAG[M_Test_GrdstFahren2]) THEN
  $FLAG[M_Test_GrdstFahren2]=TRUE
  UP_Rueckzug( )
  RETURN
ENDIF
;ENDFOLD

;-------------------------------
; Place part position
;-------------------------------
TRIGGER WHEN DISTANCE=1 DELAY=-1 DO Schrittmerker_R1Place(10034,10035,FPlace_R1_L1_S2_AP,XPlace_R1_L1_S2_AP) PRIO=-1
;FOLD LIN Place_R1_L1_S2_AP Vel=0.2 m/s LPlace_R1_L1_S2_AP Tool[2]:Lower Gripper Base[1]:Rack1;%{PE}%R8.3.21,%MKUKATPBASIS,%CMOVE,%VLIN,%P 1:LIN, 2:Place_R1_L1_S2_AP, 3:, 5:0.2, 7:LPlace_R1_L1_S2_AP
$BWDSTART=FALSE
LDAT_ACT= LLPlace_R1_L1_S2_AP
FDAT_ACT= FPlace_R1_L1_S2_AP
BAS(#CP_PARAMS,0.2)
LIN XPlace_R1_L1_S2_AP
;ENDFOLD

;FOLD Test the way back home - part 2
CONTINUE
IF $FLAG[M_Test_GrdstFahren2] THEN
  $FLAG[M_Test_GrdstFahren2]=FALSE
  UP_Rueckzug( )
  RETURN
ENDIF
;ENDFOLD

;***************************************************
; Disable part lost detection
SetPartLostDetection(NO_PART)
;***************************************************

TRIGGER WHEN DISTANCE=1 DELAY=-1 DO Schrittmerker_R1Place(10035,10036,FPlace_R1_L1_S2_NP1,XPlace_R1_L1_S2_NP1) PRIO=-1
;FOLD LIN Place_R1_L1_S2_NP1 Vel=0.2 m/s LPlace_R1_L1_S2_NP1 Tool[2]:Lower Gripper Base[1]:Rack 1 ;%{PE}
;FOLD Parameters ;%{h}
;Params IlfProvider=kukaroboter.basistech.inlineforms.movement.old; Kuka.IsGlobalPoint=False; Kuka.PointName=Place_R1_L1_S2_NP1; Kuka.BlendingEnabled=True; Kuka.MoveDataName=LPlace_R1_L1_S2_NP1; Kuka.VelocityPath=0.2; Kuka.CurrentCDSetIndex=0; Kuka.MovementParameterFieldEnabled=True; IlfCommand=LIN
;ENDFOLD
$BWDSTART = FALSE
LDAT_ACT = LLPlace_R1_L1_S2_NP1
FDAT_ACT = FPlace_R1_L1_S2_NP1
BAS(#CP_PARAMS, 0.2)
SET_CD_PARAMS (0)
LIN XPlace_R1_L1_S2_NP1
;ENDFOLD

;***************************************************
; Check for part present (empty gripper)
CheckPartPresent(EMPTY_GRIPPER)
;***************************************************
; set load data
SetLoadData( )
;***************************************************

TRIGGER WHEN DISTANCE=1 DELAY=-1 DO Schrittmerker_R1Place(10036,10037,FPlace_R1_L1_S2_NP2,XPlace_R1_L1_S2_NP2) PRIO=-1
;FOLD LIN Place_R1_L1_S2_NP2 CONT Vel=0.5 m/s LPlace_R1_L1_S2_NP2 Tool[2]:Lower Gripper Base[1]:Rack1;%{PE}%R8.3.21,%MKUKATPBASIS,%CMOVE,%VLIN,%P 1:LIN, 2:Place_R1_L1_S2_NP2, 3:C_DIS C_DIS, 5:0.5, 7:LPlace_R1_L1_S2_NP2
$BWDSTART=FALSE
LDAT_ACT= LLPlace_R1_L1_S2_NP2
FDAT_ACT= FPlace_R1_L1_S2_NP2
BAS(#CP_PARAMS,0.5)
LIN XPlace_R1_L1_S2_NP2 C_DIS C_DIS
;ENDFOLD
TRIGGER WHEN DISTANCE=1 DELAY=-1 DO Schrittmerker_R1Place(10037,10038,FPlace_R1_L1_S2_NP3,XPlace_R1_L1_S2_NP3) PRIO=-1
;FOLD LIN Place_R1_L1_S2_NP3 CONT Vel=0.5 m/s LPlace_R1_L1_S2_NP3 Tool[2]:Lower Gripper Base[1]:Rack1;%{PE}%R8.3.21,%MKUKATPBASIS,%CMOVE,%VLIN,%P 1:LIN, 2:Place_R1_L1_S2_NP3, 3:C_DIS C_DIS, 5:0.5, 7:LPlace_R1_L1_S2_NP3
$BWDSTART=FALSE
LDAT_ACT= LLPlace_R1_L1_S2_NP3
FDAT_ACT= FPlace_R1_L1_S2_NP3
BAS(#CP_PARAMS,0.5)
LIN XPlace_R1_L1_S2_NP3 C_DIS C_DIS
;ENDFOLD
TRIGGER WHEN DISTANCE=1 DELAY=-1 DO Schrittmerker_R1Place(10038,10039,FPlace_R1_L1_S2_NP4,XPlace_R1_L1_S2_NP4) PRIO=-1
;FOLD PTP Place_R1_L1_S2_NP4 CONT Vel=100 % PPlace_R1_L1_S2_NP4 Tool[2]:Lower Gripper Base[0];%{PE}%R8.3.21,%MKUKATPBASIS,%CMOVE,%VPTP,%P 1:PTP, 2:Place_R1_L1_S2_NP4, 3:C_DIS, 5:100, 7:PPlace_R1_L1_S2_NP4
$BWDSTART=FALSE
PDAT_ACT= PPPlace_R1_L1_S2_NP4
FDAT_ACT= FPlace_R1_L1_S2_NP4
BAS(#PTP_PARAMS,100)
PTP XPlace_R1_L1_S2_NP4 C_DIS
;ENDFOLD
TRIGGER WHEN DISTANCE=1 DELAY=-1 DO Schrittmerker_R1Place(10039,10040,FPlace_R1_L1_S2_NP5,XPlace_R1_L1_S2_NP5) PRIO=-1
;FOLD PTP Place_R1_L1_S2_NP5 CONT Vel=100 % PPlace_R1_L1_S2_NP5 Tool[2]:Lower Gripper Base[0];%{PE}%R8.3.21,%MKUKATPBASIS,%CMOVE,%VPTP,%P 1:PTP, 2:Place_R1_L1_S2_NP5, 3:C_DIS, 5:100, 7:PPlace_R1_L1_S2_NP5
$BWDSTART=FALSE
PDAT_ACT= PPPlace_R1_L1_S2_NP5
FDAT_ACT= FPlace_R1_L1_S2_NP5
BAS(#PTP_PARAMS,100)
PTP XPlace_R1_L1_S2_NP5 C_DIS
;ENDFOLD
TRIGGER WHEN DISTANCE=1 DELAY=-1 DO Schrittmerker_R1Place(10040,10041,FPlace_R1_L1_S2_NP6,XPlace_R1_L1_S2_NP6) PRIO=-1
;FOLD PTP Place_R1_L1_S2_NP6 CONT Vel=100 % PPlace_R1_L1_S2_NP6 Tool[2]:Lower Gripper Base[0];%{PE}%R8.3.21,%MKUKATPBASIS,%CMOVE,%VPTP,%P 1:PTP, 2:Place_R1_L1_S2_NP6, 3:C_DIS, 5:100, 7:PPlace_R1_L1_S2_NP6
$BWDSTART=FALSE
PDAT_ACT= PPPlace_R1_L1_S2_NP6
FDAT_ACT= FPlace_R1_L1_S2_NP6
BAS(#PTP_PARAMS,100)
PTP XPlace_R1_L1_S2_NP6 C_DIS
;ENDFOLD
TRIGGER WHEN DISTANCE=1 DELAY=-1 DO Schrittmerker_R1Place(10041,10042,FPlace_R1_L1_S2_NP7,XPlace_R1_L1_S2_NP7) PRIO=-1
;FOLD PTP Place_R1_L1_S2_NP7 CONT Vel=100 % PPlace_R1_L1_S2_NP7 Tool[2]:Lower Gripper Base[0];%{PE}%R8.3.21,%MKUKATPBASIS,%CMOVE,%VPTP,%P 1:PTP, 2:Place_R1_L1_S2_NP7, 3:C_DIS, 5:100, 7:PPlace_R1_L1_S2_NP7
$BWDSTART=FALSE
PDAT_ACT= PPPlace_R1_L1_S2_NP7
FDAT_ACT= FPlace_R1_L1_S2_NP7
BAS(#PTP_PARAMS,100)
PTP XPlace_R1_L1_S2_NP7 C_DIS
;ENDFOLD
TRIGGER WHEN DISTANCE=1 DELAY=-1 DO Schrittmerker_R1Place(10042,10043,FPlace_R1_L1_S2_NP8,XPlace_R1_L1_S2_NP8) PRIO=-1
;FOLD PTP Place_R1_L1_S2_NP8 CONT Vel=100 % PPlace_R1_L1_S2_NP8 Tool[2]:Lower Gripper Base[0];%{PE}%R8.3.21,%MKUKATPBASIS,%CMOVE,%VPTP,%P 1:PTP, 2:Place_R1_L1_S2_NP8, 3:C_DIS, 5:100, 7:PPlace_R1_L1_S2_NP8
$BWDSTART=FALSE
PDAT_ACT= PPPlace_R1_L1_S2_NP8
FDAT_ACT= FPlace_R1_L1_S2_NP8
BAS(#PTP_PARAMS,100)
PTP XPlace_R1_L1_S2_NP8 C_DIS
;ENDFOLD

TRIGGER WHEN DISTANCE=1 DELAY=-1 DO Schrittmerker_R1Place(10043,10002,FHOME1,$nullframe,XHOME1) PRIO=-1
;FOLD PTP HOME1 Vel=100 % PHome1;%{PE}%R8.3.21,%MKUKATPBASIS,%CMOVE,%VPTP,%P 1:PTP, 2:HOME1, 3:, 5:100, 7:PHome1
$BWDSTART=FALSE
PDAT_ACT= PPHome1
FDAT_ACT= FHOME1
BAS(#PTP_PARAMS,100)
PTP XHOME1
;ENDFOLD

;***************************************************
;FOLD Final tasks.
; Robot out of area Rack 1 Level 1
RobAusStorage1_1_A67=RESET_IN_AREA
;***************************************************
; stop cyclic clearence check
$CYCFLAG[ciFreigabeSPS]=DISABLE_MONITORING
;***************************************************
; Disable collision detection
;FOLD COLLDETECT Off ;%{PE}
;FOLD Parameters ;%{h}
;Params IlfProvider=kukaroboter.basistech.inlineforms.colldetect.off; CollDetect.Command=Off
;ENDFOLD
USE_CD_PARAMS(0)
;ENDFOLD
;***************************************************
;ENDFOLD
;***************************************************

END

; ##################################################

GLOBAL DEF UP_Place_R1_L1_S3( )
;***************************************************
; Place part on:
;    Rack  1
;    Level 1
;    Shelf 3
;***************************************************
;FOLD Preconditions - Vorraussetzungen
;***************************************************
; Enable collision detection
;FOLD COLLDETECT SetLimits Axis1: 150 % Axis2: 200 % Axis3: 150 % Axis4: 200 % Axis5: 150 % Axis6: 150 % ;%{PE}
;FOLD Parameters ;%{h}
;Params IlfProvider=kukaroboter.basistech.inlineforms.colldetect.setlimits; CollDetect.Command=SetLimits; CollDetect.Axis1=150; CollDetect.Axis2=200; CollDetect.Axis3=150; CollDetect.Axis4=200; CollDetect.Axis5=150; CollDetect.Axis6=150
;ENDFOLD
SET_TQ_VALUES(150, 200, 150, 200, 150, 150)
;ENDFOLD
;***************************************************
; Check for part in gripper (tool 2).
CheckPartPresent(OCCUPIED_GRIPPER,PART_ON_TOOL_2)
;***************************************************
; Enable part lost detection for tool 2
SetPartLostDetection(PART_ON_TOOL_2)
;***************************************************
; Set load data.
SetLoadData( )
;***************************************************
; Robot has to start from home position.
IF NOT $IN_HOME1 THEN
  UP_HomeToHome(1)
ENDIF
;***************************************************
;ENDFOLD

TRIGGER WHEN DISTANCE=1 DELAY=-1 DO Schrittmerker_R1Place(10002,10002,FHOME1,$nullframe,XHOME1) PRIO=-1
;FOLD PTP HOME1 Vel=12 % PHome1;%{PE}%R8.3.21,%MKUKATPBASIS,%CMOVE,%VPTP,%P 1:PTP, 2:HOME1, 3:, 5:12, 7:PHome1
$BWDSTART=FALSE
PDAT_ACT= PPHome1
FDAT_ACT= FHOME1
BAS(#PTP_PARAMS,12)
PTP XHOME1
;ENDFOLD

;***************************************************
;FOLD Area clearence handshake.
IF NOT $FLAG[M_Inbetriebnahme] THEN
  ;-------------------------------------------------
  ; Request area clearence.
  AnfStoer_Store1_1_A99=SET_REQUEST
  ;-------------------------------------------------
  ; Wait for area clearence from PLC.
  WAIT_FOR_INPUT("Frg_Storage1_1_E67",TRUE)
  ;-------------------------------------------------
  ; Reset area clearence request.
  AnfStoer_Store1_1_A99=RESET_REQUEST
  ;-------------------------------------------------
  ; start cyclic clearence check
  $CYCFLAG[ciFreigabeSPS]=Frg_Storage1_1_E67
  ;-------------------------------------------------
ENDIF
;***************************************************
; set "robot in area"
RobAusStorage1_1_A67=SET_IN_AREA
;ENDFOLD
;***************************************************

;***************************************************
;FOLD Check for Teachmode
IF $FLAG[M_Teachen] THEN
  WAIT FOR $T1
ENDIF
;ENDFOLD
;***************************************************

; move to the rack
TRIGGER WHEN DISTANCE=1 DELAY=-1 DO Schrittmerker_R1Place(10045,10002,FPlace_R1_L1_S3_VP1,XPlace_R1_L1_S3_VP1) PRIO=-1
;FOLD PTP Place_R1_L1_S3_VP1 CONT Vel=12 % PPlace_R1_L1_S3_VP1 Tool[2]:Lower Gripper Base[0];%{PE}%R8.3.21,%MKUKATPBASIS,%CMOVE,%VPTP,%P 1:PTP, 2:Place_R1_L1_S3_VP1, 3:C_DIS, 5:12, 7:PPlace_R1_L1_S3_VP1
$BWDSTART=FALSE
PDAT_ACT= PPPlace_R1_L1_S3_VP1
FDAT_ACT= FPlace_R1_L1_S3_VP1
BAS(#PTP_PARAMS,12)
PTP XPlace_R1_L1_S3_VP1 C_DIS
;ENDFOLD
TRIGGER WHEN DISTANCE=1 DELAY=-1 DO Schrittmerker_R1Place(10046,10045,FPlace_R1_L1_S3_VP2,XPlace_R1_L1_S3_VP2) PRIO=-1
;FOLD PTP Place_R1_L1_S3_VP2 CONT Vel=12 % PPlace_R1_L1_S3_VP2 Tool[2]:Lower Gripper Base[0];%{PE}%R8.3.21,%MKUKATPBASIS,%CMOVE,%VPTP,%P 1:PTP, 2:Place_R1_L1_S3_VP2, 3:C_DIS, 5:12, 7:PPlace_R1_L1_S3_VP2
$BWDSTART=FALSE
PDAT_ACT= PPPlace_R1_L1_S3_VP2
FDAT_ACT= FPlace_R1_L1_S3_VP2
BAS(#PTP_PARAMS,12)
PTP XPlace_R1_L1_S3_VP2 C_DIS
;ENDFOLD
TRIGGER WHEN DISTANCE=1 DELAY=-1 DO Schrittmerker_R1Place(10047,10046,FPlace_R1_L1_S3_VP3,XPlace_R1_L1_S3_VP3) PRIO=-1
;FOLD PTP Place_R1_L1_S3_VP3 CONT Vel=12 % PPlace_R1_L1_S3_VP3 Tool[2]:Lower Gripper Base[0];%{PE}%R8.3.21,%MKUKATPBASIS,%CMOVE,%VPTP,%P 1:PTP, 2:Place_R1_L1_S3_VP3, 3:C_DIS, 5:12, 7:PPlace_R1_L1_S3_VP3
$BWDSTART=FALSE
PDAT_ACT= PPPlace_R1_L1_S3_VP3
FDAT_ACT= FPlace_R1_L1_S3_VP3
BAS(#PTP_PARAMS,12)
PTP XPlace_R1_L1_S3_VP3 C_DIS
;ENDFOLD
TRIGGER WHEN DISTANCE=1 DELAY=-1 DO Schrittmerker_R1Place(10048,10047,FPlace_R1_L1_S3_VP4,XPlace_R1_L1_S3_VP4) PRIO=-1
;FOLD PTP Place_R1_L1_S3_VP4 CONT Vel=12 % PPlace_R1_L1_S3_VP4 Tool[2]:Lower Gripper Base[0];%{PE}%R8.3.21,%MKUKATPBASIS,%CMOVE,%VPTP,%P 1:PTP, 2:Place_R1_L1_S3_VP4, 3:C_DIS, 5:12, 7:PPlace_R1_L1_S3_VP4
$BWDSTART=FALSE
PDAT_ACT= PPPlace_R1_L1_S3_VP4
FDAT_ACT= FPlace_R1_L1_S3_VP4
BAS(#PTP_PARAMS,12)
PTP XPlace_R1_L1_S3_VP4 C_DIS
;ENDFOLD
TRIGGER WHEN DISTANCE=1 DELAY=-1 DO Schrittmerker_R1Place(10049,10048,FPlace_R1_L1_S3_VP5,XPlace_R1_L1_S3_VP5) PRIO=-1
;FOLD PTP Place_R1_L1_S3_VP5 CONT Vel=12 % PPlace_R1_L1_S3_VP5 Tool[2]:Lower Gripper Base[0];%{PE}%R8.3.21,%MKUKATPBASIS,%CMOVE,%VPTP,%P 1:PTP, 2:Place_R1_L1_S3_VP5, 3:C_DIS, 5:12, 7:PPlace_R1_L1_S3_VP5
$BWDSTART=FALSE
PDAT_ACT= PPPlace_R1_L1_S3_VP5
FDAT_ACT= FPlace_R1_L1_S3_VP5
BAS(#PTP_PARAMS,12)
PTP XPlace_R1_L1_S3_VP5 C_DIS
;ENDFOLD
TRIGGER WHEN DISTANCE=1 DELAY=-1 DO Schrittmerker_R1Place(10050,10049,FPlace_R1_L1_S3_VP6,XPlace_R1_L1_S3_VP6) PRIO=-1
;FOLD PTP Place_R1_L1_S3_VP6 CONT Vel=12 % PPlace_R1_L1_S3_VP6 Tool[2]:Lower Gripper Base[1]:Rack1;%{PE}%R8.3.21,%MKUKATPBASIS,%CMOVE,%VPTP,%P 1:PTP, 2:Place_R1_L1_S3_VP6, 3:C_DIS, 5:12, 7:PPlace_R1_L1_S3_VP6
$BWDSTART=FALSE
PDAT_ACT= PPPlace_R1_L1_S3_VP6
FDAT_ACT= FPlace_R1_L1_S3_VP6
BAS(#PTP_PARAMS,12)
PTP XPlace_R1_L1_S3_VP6 C_DIS
;ENDFOLD

TRIGGER WHEN DISTANCE=1 DELAY=-1 DO Schrittmerker_R1Place(10051,10050,FPlace_R1_L1_S3_Check,XPlace_R1_L1_S3_Check) PRIO=-1
;FOLD PTP Place_R1_L1_S3_Check Vel=12 % PPlace_R1_L1_S3_Check Tool[2]:Lower Gripper Base[1]:Rack1;%{PE}%R8.3.21,%MKUKATPBASIS,%CMOVE,%VPTP,%P 1:PTP, 2:Place_R1_L1_S3_Check, 3:, 5:12, 7:PPlace_R1_L1_S3_Check
$BWDSTART=FALSE
PDAT_ACT= PPPlace_R1_L1_S3_Check
FDAT_ACT= FPlace_R1_L1_S3_Check
BAS(#PTP_PARAMS,12)
PTP XPlace_R1_L1_S3_Check
;ENDFOLD

;***************************************************
;FOLD Pruefe Platz frei
IF (DetectPart(CHECK_SHELF,PLACE)==OCCUPIED) THEN
  UP_Rueckzug_R1Place( )
  RETURN
ENDIF
;ENDFOLD
;***************************************************

TRIGGER WHEN DISTANCE=1 DELAY=-1 DO Schrittmerker_R1Place(10052,10051,FPlace_R1_L1_S3_VP7,XPlace_R1_L1_S3_VP7) PRIO=-1
;FOLD LIN Place_R1_L1_S3_VP7 CONT Vel=0.5 m/s LPlace_R1_L1_S3_VP7 Tool[2]:Lower Gripper Base[1]:Rack1;%{PE}%R8.3.21,%MKUKATPBASIS,%CMOVE,%VLIN,%P 1:LIN, 2:Place_R1_L1_S3_VP7, 3:C_DIS C_DIS, 5:0.5, 7:LPlace_R1_L1_S3_VP7
$BWDSTART=FALSE
LDAT_ACT= LLPlace_R1_L1_S3_VP7
FDAT_ACT= FPlace_R1_L1_S3_VP7
BAS(#CP_PARAMS,0.5)
LIN XPlace_R1_L1_S3_VP7 C_DIS C_DIS
;ENDFOLD
TRIGGER WHEN DISTANCE=1 DELAY=-1 DO Schrittmerker_R1Place(10053,10052,FPlace_R1_L1_S3_VP8,XPlace_R1_L1_S3_VP8) PRIO=-1
;FOLD LIN Place_R1_L1_S3_VP8 CONT Vel=0.5 m/s LPlace_R1_L1_S3_VP8 Tool[2]:Lower Gripper Base[1]:Rack1;%{PE}%R8.3.21,%MKUKATPBASIS,%CMOVE,%VLIN,%P 1:LIN, 2:Place_R1_L1_S3_VP8, 3:C_DIS C_DIS, 5:0.5, 7:LPlace_R1_L1_S3_VP8
$BWDSTART=FALSE
LDAT_ACT= LLPlace_R1_L1_S3_VP8
FDAT_ACT= FPlace_R1_L1_S3_VP8
BAS(#CP_PARAMS,0.5)
LIN XPlace_R1_L1_S3_VP8 C_DIS C_DIS
;ENDFOLD

;FOLD Test the way back home - part 1
CONTINUE
IF ($FLAG[M_Test_GrdstFahren1] AND NOT $FLAG[M_Test_GrdstFahren2]) THEN
  $FLAG[M_Test_GrdstFahren2]=TRUE
  UP_Rueckzug( )
  RETURN
ENDIF
;ENDFOLD

;-------------------------------
; Place part position
;-------------------------------
TRIGGER WHEN DISTANCE=1 DELAY=-1 DO Schrittmerker_R1Place(10054,10055,FPlace_R1_L1_S3_AP,XPlace_R1_L1_S3_AP) PRIO=-1
;FOLD LIN Place_R1_L1_S3_AP Vel=0.2 m/s LPlace_R1_L1_S3_AP Tool[2]:Lower Gripper Base[1]:Rack1;%{PE}%R8.3.21,%MKUKATPBASIS,%CMOVE,%VLIN,%P 1:LIN, 2:Place_R1_L1_S3_AP, 3:, 5:0.2, 7:LPlace_R1_L1_S3_AP
$BWDSTART=FALSE
LDAT_ACT= LLPlace_R1_L1_S3_AP
FDAT_ACT= FPlace_R1_L1_S3_AP
BAS(#CP_PARAMS,0.2)
LIN XPlace_R1_L1_S3_AP
;ENDFOLD

;FOLD Test the way back home - part 2
CONTINUE
IF $FLAG[M_Test_GrdstFahren2] THEN
  $FLAG[M_Test_GrdstFahren2]=FALSE
  UP_Rueckzug( )
  RETURN
ENDIF
;ENDFOLD

;***************************************************
; Disable part lost detection
SetPartLostDetection(NO_PART)
;***************************************************

TRIGGER WHEN DISTANCE=1 DELAY=-1 DO Schrittmerker_R1Place(10055,10056,FPlace_R1_L1_S3_NP1,XPlace_R1_L1_S3_NP1) PRIO=-1
;FOLD LIN Place_R1_L1_S3_NP1 Vel=0.2 m/s LPlace_R1_L1_S3_NP1 Tool[2]:Lower Gripper Base[1]:Rack1;%{PE}%R8.3.21,%MKUKATPBASIS,%CMOVE,%VLIN,%P 1:LIN, 2:Place_R1_L1_S3_NP1, 3:C_DIS C_DIS, 5:0.2, 7:LPlace_R1_L1_S3_NP1
$BWDSTART=FALSE
LDAT_ACT= LLPlace_R1_L1_S3_NP1
FDAT_ACT= FPlace_R1_L1_S3_NP1
BAS(#CP_PARAMS,0.2)
LIN XPlace_R1_L1_S3_NP1
;ENDFOLD

;***************************************************
; Check for part present (empty gripper)
CheckPartPresent(EMPTY_GRIPPER)
;***************************************************
; set load data
SetLoadData( )
;***************************************************

TRIGGER WHEN DISTANCE=1 DELAY=-1 DO Schrittmerker_R1Place(10056,10057,FPlace_R1_L1_S3_NP2,XPlace_R1_L1_S3_NP2) PRIO=-1
;FOLD LIN Place_R1_L1_S3_NP2 CONT Vel=0.5 m/s LPlace_R1_L1_S3_NP2 Tool[2]:Lower Gripper Base[1]:Rack1;%{PE}%R8.3.21,%MKUKATPBASIS,%CMOVE,%VLIN,%P 1:LIN, 2:Place_R1_L1_S3_NP2, 3:C_DIS C_DIS, 5:0.5, 7:LPlace_R1_L1_S3_NP2
$BWDSTART=FALSE
LDAT_ACT= LLPlace_R1_L1_S3_NP2
FDAT_ACT= FPlace_R1_L1_S3_NP2
BAS(#CP_PARAMS,0.5)
LIN XPlace_R1_L1_S3_NP2 C_DIS C_DIS
;ENDFOLD
TRIGGER WHEN DISTANCE=1 DELAY=-1 DO Schrittmerker_R1Place(10057,10058,FPlace_R1_L1_S3_NP3,XPlace_R1_L1_S3_NP3) PRIO=-1
;FOLD LIN Place_R1_L1_S3_NP3 CONT Vel=0.5 m/s LPlace_R1_L1_S3_NP3 Tool[2]:Lower Gripper Base[1]:Rack1;%{PE}%R8.3.21,%MKUKATPBASIS,%CMOVE,%VLIN,%P 1:LIN, 2:Place_R1_L1_S3_NP3, 3:C_DIS C_DIS, 5:0.5, 7:LPlace_R1_L1_S3_NP3
$BWDSTART=FALSE
LDAT_ACT= LLPlace_R1_L1_S3_NP3
FDAT_ACT= FPlace_R1_L1_S3_NP3
BAS(#CP_PARAMS,0.5)
LIN XPlace_R1_L1_S3_NP3 C_DIS C_DIS
;ENDFOLD
TRIGGER WHEN DISTANCE=1 DELAY=-1 DO Schrittmerker_R1Place(10058,10059,FPlace_R1_L1_S3_NP4,XPlace_R1_L1_S3_NP4) PRIO=-1
;FOLD PTP Place_R1_L1_S3_NP4 CONT Vel=100 % PPlace_R1_L1_S3_NP4 Tool[2]:Lower Gripper Base[0];%{PE}%R8.3.21,%MKUKATPBASIS,%CMOVE,%VPTP,%P 1:PTP, 2:Place_R1_L1_S3_NP4, 3:C_DIS, 5:100, 7:PPlace_R1_L1_S3_NP4
$BWDSTART=FALSE
PDAT_ACT= PPPlace_R1_L1_S3_NP4
FDAT_ACT= FPlace_R1_L1_S3_NP4
BAS(#PTP_PARAMS,100)
PTP XPlace_R1_L1_S3_NP4 C_DIS
;ENDFOLD
TRIGGER WHEN DISTANCE=1 DELAY=-1 DO Schrittmerker_R1Place(10059,10060,FPlace_R1_L1_S3_NP5,XPlace_R1_L1_S3_NP5) PRIO=-1
;FOLD PTP Place_R1_L1_S3_NP5 CONT Vel=100 % PPlace_R1_L1_S3_NP5 Tool[2]:Lower Gripper Base[0];%{PE}%R8.3.21,%MKUKATPBASIS,%CMOVE,%VPTP,%P 1:PTP, 2:Place_R1_L1_S3_NP5, 3:C_DIS, 5:100, 7:PPlace_R1_L1_S3_NP5
$BWDSTART=FALSE
PDAT_ACT= PPPlace_R1_L1_S3_NP5
FDAT_ACT= FPlace_R1_L1_S3_NP5
BAS(#PTP_PARAMS,100)
PTP XPlace_R1_L1_S3_NP5 C_DIS
;ENDFOLD
TRIGGER WHEN DISTANCE=1 DELAY=-1 DO Schrittmerker_R1Place(10060,10061,FPlace_R1_L1_S3_NP6,XPlace_R1_L1_S3_NP6) PRIO=-1
;FOLD PTP Place_R1_L1_S3_NP6 CONT Vel=100 % PPlace_R1_L1_S3_NP6 Tool[2]:Lower Gripper Base[0];%{PE}%R8.3.21,%MKUKATPBASIS,%CMOVE,%VPTP,%P 1:PTP, 2:Place_R1_L1_S3_NP6, 3:C_DIS, 5:100, 7:PPlace_R1_L1_S3_NP6
$BWDSTART=FALSE
PDAT_ACT= PPPlace_R1_L1_S3_NP6
FDAT_ACT= FPlace_R1_L1_S3_NP6
BAS(#PTP_PARAMS,100)
PTP XPlace_R1_L1_S3_NP6 C_DIS
;ENDFOLD
TRIGGER WHEN DISTANCE=1 DELAY=-1 DO Schrittmerker_R1Place(10061,10062,FPlace_R1_L1_S3_NP7,XPlace_R1_L1_S3_NP7) PRIO=-1
;FOLD PTP Place_R1_L1_S3_NP7 CONT Vel=100 % PPlace_R1_L1_S3_NP7 Tool[2]:Lower Gripper Base[0];%{PE}%R8.3.21,%MKUKATPBASIS,%CMOVE,%VPTP,%P 1:PTP, 2:Place_R1_L1_S3_NP7, 3:C_DIS, 5:100, 7:PPlace_R1_L1_S3_NP7
$BWDSTART=FALSE
PDAT_ACT= PPPlace_R1_L1_S3_NP7
FDAT_ACT= FPlace_R1_L1_S3_NP7
BAS(#PTP_PARAMS,100)
PTP XPlace_R1_L1_S3_NP7 C_DIS
;ENDFOLD
TRIGGER WHEN DISTANCE=1 DELAY=-1 DO Schrittmerker_R1Place(10062,10063,FPlace_R1_L1_S3_NP8,XPlace_R1_L1_S3_NP8) PRIO=-1
;FOLD PTP Place_R1_L1_S3_NP8 CONT Vel=100 % PPlace_R1_L1_S3_NP8 Tool[2]:Lower Gripper Base[0];%{PE}%R8.3.21,%MKUKATPBASIS,%CMOVE,%VPTP,%P 1:PTP, 2:Place_R1_L1_S3_NP8, 3:C_DIS, 5:100, 7:PPlace_R1_L1_S3_NP8
$BWDSTART=FALSE
PDAT_ACT= PPPlace_R1_L1_S3_NP8
FDAT_ACT= FPlace_R1_L1_S3_NP8
BAS(#PTP_PARAMS,100)
PTP XPlace_R1_L1_S3_NP8 C_DIS
;ENDFOLD

TRIGGER WHEN DISTANCE=1 DELAY=-1 DO Schrittmerker_R1Place(10063,10002,FHOME1,$nullframe,XHOME1) PRIO=-1
;FOLD PTP HOME1 Vel=100 % PHome1;%{PE}%R8.3.21,%MKUKATPBASIS,%CMOVE,%VPTP,%P 1:PTP, 2:HOME1, 3:, 5:100, 7:PHome1
$BWDSTART=FALSE
PDAT_ACT= PPHome1
FDAT_ACT= FHOME1
BAS(#PTP_PARAMS,100)
PTP XHOME1
;ENDFOLD

;***************************************************
;FOLD Final tasks.
; Robot out of area Rack 1 Level 1
RobAusStorage1_1_A67=RESET_IN_AREA
;***************************************************
; stop cyclic clearence check
$CYCFLAG[ciFreigabeSPS]=DISABLE_MONITORING
;***************************************************
; Disable collision detection
;FOLD COLLDETECT Off ;%{PE}
;FOLD Parameters ;%{h}
;Params IlfProvider=kukaroboter.basistech.inlineforms.colldetect.off; CollDetect.Command=Off
;ENDFOLD
USE_CD_PARAMS(0)
;ENDFOLD
;***************************************************
;ENDFOLD
;***************************************************

END

; ##################################################

GLOBAL DEF UP_Place_R1_L1_S4( )
;***************************************************
; Place part on:
;    Rack  1
;    Level 1
;    Shelf 4
;***************************************************
;FOLD Preconditions - Vorraussetzungen
;***************************************************
; Enable collision detection
;FOLD COLLDETECT SetLimits Axis1: 150 % Axis2: 200 % Axis3: 150 % Axis4: 200 % Axis5: 150 % Axis6: 150 % ;%{PE}
;FOLD Parameters ;%{h}
;Params IlfProvider=kukaroboter.basistech.inlineforms.colldetect.setlimits; CollDetect.Command=SetLimits; CollDetect.Axis1=150; CollDetect.Axis2=200; CollDetect.Axis3=150; CollDetect.Axis4=200; CollDetect.Axis5=150; CollDetect.Axis6=150
;ENDFOLD
SET_TQ_VALUES(150, 200, 150, 200, 150, 150)
;ENDFOLD
;***************************************************
; Check for part in gripper (tool 2).
CheckPartPresent(OCCUPIED_GRIPPER,PART_ON_TOOL_2)
;***************************************************
; Enable part lost detection for tool 2
SetPartLostDetection(PART_ON_TOOL_2)
;***************************************************
; Set load data.
SetLoadData( )
;***************************************************
; Robot has to start from home position.
IF NOT $IN_HOME1 THEN
  UP_HomeToHome(1)
ENDIF
;***************************************************
;ENDFOLD

TRIGGER WHEN DISTANCE=1 DELAY=-1 DO Schrittmerker_R1Place(10002,10002,FHOME1,$nullframe,XHOME1) PRIO=-1
;FOLD PTP HOME1 Vel=12 % PHome1;%{PE}%R8.3.21,%MKUKATPBASIS,%CMOVE,%VPTP,%P 1:PTP, 2:HOME1, 3:, 5:12, 7:PHome1
$BWDSTART=FALSE
PDAT_ACT= PPHome1
FDAT_ACT= FHOME1
BAS(#PTP_PARAMS,12)
PTP XHOME1
;ENDFOLD

;***************************************************
;FOLD Area clearence handshake.
IF NOT $FLAG[M_Inbetriebnahme] THEN
  ;-------------------------------------------------
  ; Request area clearence.
  AnfStoer_Store1_1_A99=SET_REQUEST
  ;-------------------------------------------------
  ; Wait for area clearence from PLC.
  WAIT_FOR_INPUT("Frg_Storage1_1_E67",TRUE)
  ;-------------------------------------------------
  ; Reset area clearence request.
  AnfStoer_Store1_1_A99=RESET_REQUEST
  ;-------------------------------------------------
  ; start cyclic clearence check
  $CYCFLAG[ciFreigabeSPS]=Frg_Storage1_1_E67
  ;-------------------------------------------------
ENDIF
;***************************************************
; set "robot in area"
RobAusStorage1_1_A67=SET_IN_AREA
;ENDFOLD
;***************************************************

;***************************************************
;FOLD Check for Teachmode
IF $FLAG[M_Teachen] THEN
  WAIT FOR $T1
ENDIF
;ENDFOLD
;***************************************************

; move to the rack
TRIGGER WHEN DISTANCE=1 DELAY=-1 DO Schrittmerker_R1Place(10065,10002,FPlace_R1_L1_S4_VP1,XPlace_R1_L1_S4_VP1) PRIO=-1
;FOLD PTP Place_R1_L1_S4_VP1 CONT Vel=12 % PPlace_R1_L1_S4_VP1 Tool[2]:Lower Gripper Base[0];%{PE}%R8.3.21,%MKUKATPBASIS,%CMOVE,%VPTP,%P 1:PTP, 2:Place_R1_L1_S4_VP1, 3:C_DIS, 5:12, 7:PPlace_R1_L1_S4_VP1
$BWDSTART=FALSE
PDAT_ACT= PPPlace_R1_L1_S4_VP1
FDAT_ACT= FPlace_R1_L1_S4_VP1
BAS(#PTP_PARAMS,12)
PTP XPlace_R1_L1_S4_VP1 C_DIS
;ENDFOLD
TRIGGER WHEN DISTANCE=1 DELAY=-1 DO Schrittmerker_R1Place(10066,10065,FPlace_R1_L1_S4_VP2,XPlace_R1_L1_S4_VP2) PRIO=-1
;FOLD PTP Place_R1_L1_S4_VP2 CONT Vel=12 % PPlace_R1_L1_S4_VP2 Tool[2]:Lower Gripper Base[0];%{PE}%R8.3.21,%MKUKATPBASIS,%CMOVE,%VPTP,%P 1:PTP, 2:Place_R1_L1_S4_VP2, 3:C_DIS, 5:12, 7:PPlace_R1_L1_S4_VP2
$BWDSTART=FALSE
PDAT_ACT= PPPlace_R1_L1_S4_VP2
FDAT_ACT= FPlace_R1_L1_S4_VP2
BAS(#PTP_PARAMS,12)
PTP XPlace_R1_L1_S4_VP2 C_DIS
;ENDFOLD
TRIGGER WHEN DISTANCE=1 DELAY=-1 DO Schrittmerker_R1Place(10067,10066,FPlace_R1_L1_S4_VP3,XPlace_R1_L1_S4_VP3) PRIO=-1
;FOLD PTP Place_R1_L1_S4_VP3 CONT Vel=12 % PPlace_R1_L1_S4_VP3 Tool[2]:Lower Gripper Base[0];%{PE}%R8.3.21,%MKUKATPBASIS,%CMOVE,%VPTP,%P 1:PTP, 2:Place_R1_L1_S4_VP3, 3:C_DIS, 5:12, 7:PPlace_R1_L1_S4_VP3
$BWDSTART=FALSE
PDAT_ACT= PPPlace_R1_L1_S4_VP3
FDAT_ACT= FPlace_R1_L1_S4_VP3
BAS(#PTP_PARAMS,12)
PTP XPlace_R1_L1_S4_VP3 C_DIS
;ENDFOLD
TRIGGER WHEN DISTANCE=1 DELAY=-1 DO Schrittmerker_R1Place(10068,10067,FPlace_R1_L1_S4_VP4,XPlace_R1_L1_S4_VP4) PRIO=-1
;FOLD PTP Place_R1_L1_S4_VP4 CONT Vel=12 % PPlace_R1_L1_S4_VP4 Tool[2]:Lower Gripper Base[0];%{PE}%R8.3.21,%MKUKATPBASIS,%CMOVE,%VPTP,%P 1:PTP, 2:Place_R1_L1_S4_VP4, 3:C_DIS, 5:12, 7:PPlace_R1_L1_S4_VP4
$BWDSTART=FALSE
PDAT_ACT= PPPlace_R1_L1_S4_VP4
FDAT_ACT= FPlace_R1_L1_S4_VP4
BAS(#PTP_PARAMS,12)
PTP XPlace_R1_L1_S4_VP4 C_DIS
;ENDFOLD
TRIGGER WHEN DISTANCE=1 DELAY=-1 DO Schrittmerker_R1Place(10069,10068,FPlace_R1_L1_S4_VP5,XPlace_R1_L1_S4_VP5) PRIO=-1
;FOLD PTP Place_R1_L1_S4_VP5 CONT Vel=12 % PPlace_R1_L1_S4_VP5 Tool[2]:Lower Gripper Base[0];%{PE}%R8.3.21,%MKUKATPBASIS,%CMOVE,%VPTP,%P 1:PTP, 2:Place_R1_L1_S4_VP5, 3:C_DIS, 5:12, 7:PPlace_R1_L1_S4_VP5
$BWDSTART=FALSE
PDAT_ACT= PPPlace_R1_L1_S4_VP5
FDAT_ACT= FPlace_R1_L1_S4_VP5
BAS(#PTP_PARAMS,12)
PTP XPlace_R1_L1_S4_VP5 C_DIS
;ENDFOLD
TRIGGER WHEN DISTANCE=1 DELAY=-1 DO Schrittmerker_R1Place(10070,10069,FPlace_R1_L1_S4_VP6,XPlace_R1_L1_S4_VP6) PRIO=-1
;FOLD PTP Place_R1_L1_S4_VP6 CONT Vel=12 % PPlace_R1_L1_S4_VP6 Tool[2]:Lower Gripper Base[1]:Rack1;%{PE}%R8.3.21,%MKUKATPBASIS,%CMOVE,%VPTP,%P 1:PTP, 2:Place_R1_L1_S4_VP6, 3:C_DIS, 5:12, 7:PPlace_R1_L1_S4_VP6
$BWDSTART=FALSE
PDAT_ACT= PPPlace_R1_L1_S4_VP6
FDAT_ACT= FPlace_R1_L1_S4_VP6
BAS(#PTP_PARAMS,12)
PTP XPlace_R1_L1_S4_VP6 C_DIS
;ENDFOLD

TRIGGER WHEN DISTANCE=1 DELAY=-1 DO Schrittmerker_R1Place(10071,10070,FPlace_R1_L1_S4_Check,XPlace_R1_L1_S4_Check) PRIO=-1
;FOLD PTP Place_R1_L1_S4_Check Vel=12 % PPlace_R1_L1_S4_Check Tool[2]:Lower Gripper Base[1]:Rack1;%{PE}%R8.3.21,%MKUKATPBASIS,%CMOVE,%VPTP,%P 1:PTP, 2:Place_R1_L1_S4_Check, 3:, 5:12, 7:PPlace_R1_L1_S4_Check
$BWDSTART=FALSE
PDAT_ACT= PPPlace_R1_L1_S4_Check
FDAT_ACT= FPlace_R1_L1_S4_Check
BAS(#PTP_PARAMS,12)
PTP XPlace_R1_L1_S4_Check
;ENDFOLD

;***************************************************
;FOLD Pruefe Platz frei
IF (DetectPart(CHECK_SHELF,PLACE)==OCCUPIED) THEN
  UP_Rueckzug_R1Place( )
  RETURN
ENDIF
;ENDFOLD
;***************************************************

TRIGGER WHEN DISTANCE=1 DELAY=-1 DO Schrittmerker_R1Place(10072,10071,FPlace_R1_L1_S4_VP7,XPlace_R1_L1_S4_VP7) PRIO=-1
;FOLD LIN Place_R1_L1_S4_VP7 CONT Vel=0.5 m/s LPlace_R1_L1_S4_VP7 Tool[2]:Lower Gripper Base[1]:Rack1;%{PE}%R8.3.21,%MKUKATPBASIS,%CMOVE,%VLIN,%P 1:LIN, 2:Place_R1_L1_S4_VP7, 3:C_DIS C_DIS, 5:0.5, 7:LPlace_R1_L1_S4_VP7
$BWDSTART=FALSE
LDAT_ACT= LLPlace_R1_L1_S4_VP7
FDAT_ACT= FPlace_R1_L1_S4_VP7
BAS(#CP_PARAMS,0.5)
LIN XPlace_R1_L1_S4_VP7 C_DIS C_DIS
;ENDFOLD
TRIGGER WHEN DISTANCE=1 DELAY=-1 DO Schrittmerker_R1Place(10073,10072,FPlace_R1_L1_S4_VP8,XPlace_R1_L1_S4_VP8) PRIO=-1
;FOLD LIN Place_R1_L1_S4_VP8 CONT Vel=0.5 m/s LPlace_R1_L1_S4_VP8 Tool[2]:Lower Gripper Base[1]:Rack1;%{PE}%R8.3.21,%MKUKATPBASIS,%CMOVE,%VLIN,%P 1:LIN, 2:Place_R1_L1_S4_VP8, 3:C_DIS C_DIS, 5:0.5, 7:LPlace_R1_L1_S4_VP8
$BWDSTART=FALSE
LDAT_ACT= LLPlace_R1_L1_S4_VP8
FDAT_ACT= FPlace_R1_L1_S4_VP8
BAS(#CP_PARAMS,0.5)
LIN XPlace_R1_L1_S4_VP8 C_DIS C_DIS
;ENDFOLD

;FOLD Test the way back home - part 1
CONTINUE
IF ($FLAG[M_Test_GrdstFahren1] AND NOT $FLAG[M_Test_GrdstFahren2]) THEN
  $FLAG[M_Test_GrdstFahren2]=TRUE
  UP_Rueckzug( )
  RETURN
ENDIF
;ENDFOLD

;-------------------------------
; Place part position
;-------------------------------
TRIGGER WHEN DISTANCE=1 DELAY=-1 DO Schrittmerker_R1Place(10074,10075,FPlace_R1_L1_S4_AP,XPlace_R1_L1_S4_AP) PRIO=-1
;FOLD LIN Place_R1_L1_S4_AP Vel=0.2 m/s LPlace_R1_L1_S4_AP Tool[2]:Lower Gripper Base[1]:Rack1;%{PE}%R8.3.21,%MKUKATPBASIS,%CMOVE,%VLIN,%P 1:LIN, 2:Place_R1_L1_S4_AP, 3:, 5:0.2, 7:LPlace_R1_L1_S4_AP
$BWDSTART=FALSE
LDAT_ACT= LLPlace_R1_L1_S4_AP
FDAT_ACT= FPlace_R1_L1_S4_AP
BAS(#CP_PARAMS,0.2)
LIN XPlace_R1_L1_S4_AP
;ENDFOLD

;FOLD Test the way back home - part 2
CONTINUE
IF $FLAG[M_Test_GrdstFahren2] THEN
  $FLAG[M_Test_GrdstFahren2]=FALSE
  UP_Rueckzug( )
  RETURN
ENDIF
;ENDFOLD

;***************************************************
; Disable part lost detection
SetPartLostDetection(NO_PART)
;***************************************************

TRIGGER WHEN DISTANCE=1 DELAY=-1 DO Schrittmerker_R1Place(10075,10076,FPlace_R1_L1_S4_NP1,XPlace_R1_L1_S4_NP1) PRIO=-1
;FOLD LIN Place_R1_L1_S4_NP1 Vel=0.2 m/s LPlace_R1_L1_S4_NP1 Tool[2]:Lower Gripper Base[1]:Rack 1 ;%{PE}
;FOLD Parameters ;%{h}
;Params IlfProvider=kukaroboter.basistech.inlineforms.movement.old; Kuka.IsGlobalPoint=False; Kuka.PointName=Place_R1_L1_S4_NP1; Kuka.BlendingEnabled=False; Kuka.MoveDataName=LPlace_R1_L1_S4_NP1; Kuka.VelocityPath=0.2; Kuka.CurrentCDSetIndex=0; Kuka.MovementParameterFieldEnabled=True; IlfCommand=LIN
;ENDFOLD
$BWDSTART = FALSE
LDAT_ACT = LLPlace_R1_L1_S4_NP1
FDAT_ACT = FPlace_R1_L1_S4_NP1
BAS(#CP_PARAMS, 0.2)
SET_CD_PARAMS (0)
LIN XPlace_R1_L1_S4_NP1
;ENDFOLD

;***************************************************
; Check for part present (empty gripper)
CheckPartPresent(EMPTY_GRIPPER)
;***************************************************
; set load data
SetLoadData( )
;***************************************************

TRIGGER WHEN DISTANCE=1 DELAY=-1 DO Schrittmerker_R1Place(10076,10077,FPlace_R1_L1_S4_NP2,XPlace_R1_L1_S4_NP2) PRIO=-1
;FOLD LIN Place_R1_L1_S4_NP2 CONT Vel=0.5 m/s LPlace_R1_L1_S4_NP2 Tool[2]:Lower Gripper Base[1]:Rack1;%{PE}%R8.3.21,%MKUKATPBASIS,%CMOVE,%VLIN,%P 1:LIN, 2:Place_R1_L1_S4_NP2, 3:C_DIS C_DIS, 5:0.5, 7:LPlace_R1_L1_S4_NP2
$BWDSTART=FALSE
LDAT_ACT= LLPlace_R1_L1_S4_NP2
FDAT_ACT= FPlace_R1_L1_S4_NP2
BAS(#CP_PARAMS,0.5)
LIN XPlace_R1_L1_S4_NP2 C_DIS C_DIS
;ENDFOLD
TRIGGER WHEN DISTANCE=1 DELAY=-1 DO Schrittmerker_R1Place(10077,10078,FPlace_R1_L1_S4_NP3,XPlace_R1_L1_S4_NP3) PRIO=-1
;FOLD LIN Place_R1_L1_S4_NP3 CONT Vel=0.5 m/s LPlace_R1_L1_S4_NP3 Tool[2]:Lower Gripper Base[1]:Rack1;%{PE}%R8.3.21,%MKUKATPBASIS,%CMOVE,%VLIN,%P 1:LIN, 2:Place_R1_L1_S4_NP3, 3:C_DIS C_DIS, 5:0.5, 7:LPlace_R1_L1_S4_NP3
$BWDSTART=FALSE
LDAT_ACT= LLPlace_R1_L1_S4_NP3
FDAT_ACT= FPlace_R1_L1_S4_NP3
BAS(#CP_PARAMS,0.5)
LIN XPlace_R1_L1_S4_NP3 C_DIS C_DIS
;ENDFOLD
TRIGGER WHEN DISTANCE=1 DELAY=-1 DO Schrittmerker_R1Place(10078,10079,FPlace_R1_L1_S4_NP4,XPlace_R1_L1_S4_NP4) PRIO=-1
;FOLD PTP Place_R1_L1_S4_NP4 CONT Vel=100 % PPlace_R1_L1_S4_NP4 Tool[2]:Lower Gripper Base[0];%{PE}%R8.3.21,%MKUKATPBASIS,%CMOVE,%VPTP,%P 1:PTP, 2:Place_R1_L1_S4_NP4, 3:C_DIS, 5:100, 7:PPlace_R1_L1_S4_NP4
$BWDSTART=FALSE
PDAT_ACT= PPPlace_R1_L1_S4_NP4
FDAT_ACT= FPlace_R1_L1_S4_NP4
BAS(#PTP_PARAMS,100)
PTP XPlace_R1_L1_S4_NP4 C_DIS
;ENDFOLD
TRIGGER WHEN DISTANCE=1 DELAY=-1 DO Schrittmerker_R1Place(10079,10080,FPlace_R1_L1_S4_NP5,XPlace_R1_L1_S4_NP5) PRIO=-1
;FOLD PTP Place_R1_L1_S4_NP5 CONT Vel=100 % PPlace_R1_L1_S4_NP5 Tool[2]:Lower Gripper Base[0];%{PE}%R8.3.21,%MKUKATPBASIS,%CMOVE,%VPTP,%P 1:PTP, 2:Place_R1_L1_S4_NP5, 3:C_DIS, 5:100, 7:PPlace_R1_L1_S4_NP5
$BWDSTART=FALSE
PDAT_ACT= PPPlace_R1_L1_S4_NP5
FDAT_ACT= FPlace_R1_L1_S4_NP5
BAS(#PTP_PARAMS,100)
PTP XPlace_R1_L1_S4_NP5 C_DIS
;ENDFOLD
TRIGGER WHEN DISTANCE=1 DELAY=-1 DO Schrittmerker_R1Place(10080,10081,FPlace_R1_L1_S4_NP6,XPlace_R1_L1_S4_NP6) PRIO=-1
;FOLD PTP Place_R1_L1_S4_NP6 CONT Vel=100 % PPlace_R1_L1_S4_NP6 Tool[2]:Lower Gripper Base[0];%{PE}%R8.3.21,%MKUKATPBASIS,%CMOVE,%VPTP,%P 1:PTP, 2:Place_R1_L1_S4_NP6, 3:C_DIS, 5:100, 7:PPlace_R1_L1_S4_NP6
$BWDSTART=FALSE
PDAT_ACT= PPPlace_R1_L1_S4_NP6
FDAT_ACT= FPlace_R1_L1_S4_NP6
BAS(#PTP_PARAMS,100)
PTP XPlace_R1_L1_S4_NP6 C_DIS
;ENDFOLD
TRIGGER WHEN DISTANCE=1 DELAY=-1 DO Schrittmerker_R1Place(10081,10082,FPlace_R1_L1_S4_NP7,XPlace_R1_L1_S4_NP7) PRIO=-1
;FOLD PTP Place_R1_L1_S4_NP7 CONT Vel=100 % PPlace_R1_L1_S4_NP7 Tool[2]:Lower Gripper Base[0];%{PE}%R8.3.21,%MKUKATPBASIS,%CMOVE,%VPTP,%P 1:PTP, 2:Place_R1_L1_S4_NP7, 3:C_DIS, 5:100, 7:PPlace_R1_L1_S4_NP7
$BWDSTART=FALSE
PDAT_ACT= PPPlace_R1_L1_S4_NP7
FDAT_ACT= FPlace_R1_L1_S4_NP7
BAS(#PTP_PARAMS,100)
PTP XPlace_R1_L1_S4_NP7 C_DIS
;ENDFOLD
TRIGGER WHEN DISTANCE=1 DELAY=-1 DO Schrittmerker_R1Place(10082,10083,FPlace_R1_L1_S4_NP8,XPlace_R1_L1_S4_NP8) PRIO=-1
;FOLD PTP Place_R1_L1_S4_NP8 CONT Vel=100 % PPlace_R1_L1_S4_NP8 Tool[2]:Lower Gripper Base[0];%{PE}%R8.3.21,%MKUKATPBASIS,%CMOVE,%VPTP,%P 1:PTP, 2:Place_R1_L1_S4_NP8, 3:C_DIS, 5:100, 7:PPlace_R1_L1_S4_NP8
$BWDSTART=FALSE
PDAT_ACT= PPPlace_R1_L1_S4_NP8
FDAT_ACT= FPlace_R1_L1_S4_NP8
BAS(#PTP_PARAMS,100)
PTP XPlace_R1_L1_S4_NP8 C_DIS
;ENDFOLD

TRIGGER WHEN DISTANCE=1 DELAY=-1 DO Schrittmerker_R1Place(10083,10002,FHOME1,$nullframe,XHOME1) PRIO=-1
;FOLD PTP HOME1 Vel=100 % PHome1;%{PE}%R8.3.21,%MKUKATPBASIS,%CMOVE,%VPTP,%P 1:PTP, 2:HOME1, 3:, 5:100, 7:PHome1
$BWDSTART=FALSE
PDAT_ACT= PPHome1
FDAT_ACT= FHOME1
BAS(#PTP_PARAMS,100)
PTP XHOME1
;ENDFOLD

;***************************************************
;FOLD Final tasks.
; Robot out of area Rack 1 Level 1
RobAusStorage1_1_A67=RESET_IN_AREA
;***************************************************
; stop cyclic clearence check
$CYCFLAG[ciFreigabeSPS]=DISABLE_MONITORING
;***************************************************
; Disable collision detection
;FOLD COLLDETECT Off ;%{PE}
;FOLD Parameters ;%{h}
;Params IlfProvider=kukaroboter.basistech.inlineforms.colldetect.off; CollDetect.Command=Off
;ENDFOLD
USE_CD_PARAMS(0)
;ENDFOLD
;***************************************************
;ENDFOLD
;***************************************************

END

; ##################################################

GLOBAL DEF UP_Place_R1_L2_S1( )
;***************************************************
; Place part on:
;    Rack  1
;    Level 2
;    Shelf 1
;  RBG Kollision beachten!
;***************************************************
;FOLD Preconditions - Vorraussetzungen
;***************************************************
; Enable collision detection
;FOLD COLLDETECT SetLimits Axis1: 150 % Axis2: 200 % Axis3: 150 % Axis4: 200 % Axis5: 150 % Axis6: 150 % ;%{PE}
;FOLD Parameters ;%{h}
;Params IlfProvider=kukaroboter.basistech.inlineforms.colldetect.setlimits; CollDetect.Command=SetLimits; CollDetect.Axis1=150; CollDetect.Axis2=200; CollDetect.Axis3=150; CollDetect.Axis4=200; CollDetect.Axis5=150; CollDetect.Axis6=150
;ENDFOLD
SET_TQ_VALUES(150, 200, 150, 200, 150, 150)
;ENDFOLD
;***************************************************
; Check for part in gripper (tool 2).
CheckPartPresent(OCCUPIED_GRIPPER,PART_ON_TOOL_2)
;***************************************************
; Enable part lost detection for tool 2
SetPartLostDetection(PART_ON_TOOL_2)
;***************************************************
; Set load data.
SetLoadData( )
;***************************************************
; Robot has to start from home position.
IF NOT $IN_HOME1 THEN
  UP_HomeToHome(1)
ENDIF
;***************************************************
;ENDFOLD

TRIGGER WHEN DISTANCE=1 DELAY=-1 DO Schrittmerker_R1Place(10002,10002,FHOME1,$nullframe,XHOME1) PRIO=-1
;FOLD PTP HOME1 Vel=12 % PHome1;%{PE}%R8.3.21,%MKUKATPBASIS,%CMOVE,%VPTP,%P 1:PTP, 2:HOME1, 3:, 5:12, 7:PHome1
$BWDSTART=FALSE
PDAT_ACT= PPHome1
FDAT_ACT= FHOME1
BAS(#PTP_PARAMS,12)
PTP XHOME1
;ENDFOLD

;***************************************************
;FOLD Area clearence handshake.
IF NOT $FLAG[M_Inbetriebnahme] THEN
  ;-------------------------------------------------
  ; Request area clearence.
  AnfStoer_Store1_2_A100=SET_REQUEST
  ;-------------------------------------------------
  ; Wait for area clearence from PLC.
  WAIT_FOR_INPUT("Frg_Storage1_2_E68",TRUE)
  ;-------------------------------------------------
  ; Reset area clearence request.
  AnfStoer_Store1_2_A100=RESET_REQUEST
  ;-------------------------------------------------
  ; start cyclic clearence check
  $CYCFLAG[ciFreigabeSPS]=Frg_Storage1_2_E68
  ;-------------------------------------------------
ENDIF
;***************************************************
; set "robot in area"
RobAusStorage1_2_A68=SET_IN_AREA
;ENDFOLD
;***************************************************

;***************************************************
;FOLD Check for Teachmode
IF $FLAG[M_Teachen] THEN
  WAIT FOR $T1
ENDIF
;ENDFOLD
;***************************************************

; move to the rack
TRIGGER WHEN DISTANCE=1 DELAY=-1 DO Schrittmerker_R1Place(10085,10002,FPlace_R1_L2_S1_VP1,XPlace_R1_L2_S1_VP1) PRIO=-1
;FOLD PTP Place_R1_L2_S1_VP1 CONT Vel=12 % PPlace_R1_L2_S1_VP1 Tool[2]:Lower Gripper Base[0];%{PE}%R8.3.21,%MKUKATPBASIS,%CMOVE,%VPTP,%P 1:PTP, 2:Place_R1_L2_S1_VP1, 3:C_DIS, 5:12, 7:PPlace_R1_L2_S1_VP1
$BWDSTART=FALSE
PDAT_ACT= PPPlace_R1_L2_S1_VP1
FDAT_ACT= FPlace_R1_L2_S1_VP1
BAS(#PTP_PARAMS,12)
PTP XPlace_R1_L2_S1_VP1 C_DIS
;ENDFOLD
TRIGGER WHEN DISTANCE=1 DELAY=-1 DO Schrittmerker_R1Place(10086,10085,FPlace_R1_L2_S1_VP2,XPlace_R1_L2_S1_VP2) PRIO=-1
;FOLD PTP Place_R1_L2_S1_VP2 CONT Vel=12 % PPlace_R1_L2_S1_VP2 Tool[2]:Lower Gripper Base[0];%{PE}%R8.3.21,%MKUKATPBASIS,%CMOVE,%VPTP,%P 1:PTP, 2:Place_R1_L2_S1_VP2, 3:C_DIS, 5:12, 7:PPlace_R1_L2_S1_VP2
$BWDSTART=FALSE
PDAT_ACT= PPPlace_R1_L2_S1_VP2
FDAT_ACT= FPlace_R1_L2_S1_VP2
BAS(#PTP_PARAMS,12)
PTP XPlace_R1_L2_S1_VP2 C_DIS
;ENDFOLD
TRIGGER WHEN DISTANCE=1 DELAY=-1 DO Schrittmerker_R1Place(10087,10086,FPlace_R1_L2_S1_VP3,XPlace_R1_L2_S1_VP3) PRIO=-1
;FOLD PTP Place_R1_L2_S1_VP3 CONT Vel=12 % PPlace_R1_L2_S1_VP3 Tool[2]:Lower Gripper Base[0];%{PE}%R8.3.21,%MKUKATPBASIS,%CMOVE,%VPTP,%P 1:PTP, 2:Place_R1_L2_S1_VP3, 3:C_DIS, 5:12, 7:PPlace_R1_L2_S1_VP3
$BWDSTART=FALSE
PDAT_ACT= PPPlace_R1_L2_S1_VP3
FDAT_ACT= FPlace_R1_L2_S1_VP3
BAS(#PTP_PARAMS,12)
PTP XPlace_R1_L2_S1_VP3 C_DIS
;ENDFOLD
TRIGGER WHEN DISTANCE=1 DELAY=-1 DO Schrittmerker_R1Place(10088,10087,FPlace_R1_L2_S1_VP4,XPlace_R1_L2_S1_VP4) PRIO=-1
;FOLD PTP Place_R1_L2_S1_VP4 CONT Vel=12 % PPlace_R1_L2_S1_VP4 Tool[2]:Lower Gripper Base[0];%{PE}%R8.3.21,%MKUKATPBASIS,%CMOVE,%VPTP,%P 1:PTP, 2:Place_R1_L2_S1_VP4, 3:C_DIS, 5:12, 7:PPlace_R1_L2_S1_VP4
$BWDSTART=FALSE
PDAT_ACT= PPPlace_R1_L2_S1_VP4
FDAT_ACT= FPlace_R1_L2_S1_VP4
BAS(#PTP_PARAMS,12)
PTP XPlace_R1_L2_S1_VP4 C_DIS
;ENDFOLD
TRIGGER WHEN DISTANCE=1 DELAY=-1 DO Schrittmerker_R1Place(10089,10088,FPlace_R1_L2_S1_VP5,XPlace_R1_L2_S1_VP5) PRIO=-1
;FOLD PTP Place_R1_L2_S1_VP5 CONT Vel=12 % PPlace_R1_L2_S1_VP5 Tool[2]:Lower Gripper Base[0];%{PE}%R8.3.21,%MKUKATPBASIS,%CMOVE,%VPTP,%P 1:PTP, 2:Place_R1_L2_S1_VP5, 3:C_DIS, 5:12, 7:PPlace_R1_L2_S1_VP5
$BWDSTART=FALSE
PDAT_ACT= PPPlace_R1_L2_S1_VP5
FDAT_ACT= FPlace_R1_L2_S1_VP5
BAS(#PTP_PARAMS,12)
PTP XPlace_R1_L2_S1_VP5 C_DIS
;ENDFOLD
TRIGGER WHEN DISTANCE=1 DELAY=-1 DO Schrittmerker_R1Place(10090,10089,FPlace_R1_L2_S1_VP6,XPlace_R1_L2_S1_VP6) PRIO=-1
;FOLD PTP Place_R1_L2_S1_VP6 CONT Vel=12 % PPlace_R1_L2_S1_VP6 Tool[2]:Lower Gripper Base[1]:Rack1;%{PE}%R8.3.21,%MKUKATPBASIS,%CMOVE,%VPTP,%P 1:PTP, 2:Place_R1_L2_S1_VP6, 3:C_DIS, 5:12, 7:PPlace_R1_L2_S1_VP6
$BWDSTART=FALSE
PDAT_ACT= PPPlace_R1_L2_S1_VP6
FDAT_ACT= FPlace_R1_L2_S1_VP6
BAS(#PTP_PARAMS,12)
PTP XPlace_R1_L2_S1_VP6 C_DIS
;ENDFOLD

TRIGGER WHEN DISTANCE=1 DELAY=-1 DO Schrittmerker_R1Place(10091,10090,FPlace_R1_L2_S1_Check,XPlace_R1_L2_S1_Check) PRIO=-1
;FOLD PTP Place_R1_L2_S1_Check Vel=12 % PPlace_R1_L2_S1_Check Tool[2]:Lower Gripper Base[1]:Rack1;%{PE}%R8.3.21,%MKUKATPBASIS,%CMOVE,%VPTP,%P 1:PTP, 2:Place_R1_L2_S1_Check, 3:, 5:12, 7:PPlace_R1_L2_S1_Check
$BWDSTART=FALSE
PDAT_ACT= PPPlace_R1_L2_S1_Check
FDAT_ACT= FPlace_R1_L2_S1_Check
BAS(#PTP_PARAMS,12)
PTP XPlace_R1_L2_S1_Check
;ENDFOLD

;***************************************************
;FOLD Pruefe Platz frei
IF (DetectPart(CHECK_SHELF,PLACE)==OCCUPIED) THEN
  UP_Rueckzug_R1Place( )
  RETURN
ENDIF
;ENDFOLD
;***************************************************

TRIGGER WHEN DISTANCE=1 DELAY=-1 DO Schrittmerker_R1Place(10092,10091,FPlace_R1_L2_S1_VP7,XPlace_R1_L2_S1_VP7) PRIO=-1
;FOLD LIN Place_R1_L2_S1_VP7 CONT Vel=0.5 m/s LPlace_R1_L2_S1_VP7 Tool[2]:Lower Gripper Base[1]:Rack1;%{PE}%R8.3.21,%MKUKATPBASIS,%CMOVE,%VLIN,%P 1:LIN, 2:Place_R1_L2_S1_VP7, 3:C_DIS C_DIS, 5:0.5, 7:LPlace_R1_L2_S1_VP7
$BWDSTART=FALSE
LDAT_ACT= LLPlace_R1_L2_S1_VP7
FDAT_ACT= FPlace_R1_L2_S1_VP7
BAS(#CP_PARAMS,0.5)
LIN XPlace_R1_L2_S1_VP7 C_DIS C_DIS
;ENDFOLD
TRIGGER WHEN DISTANCE=1 DELAY=-1 DO Schrittmerker_R1Place(10093,10092,FPlace_R1_L2_S1_VP8,XPlace_R1_L2_S1_VP8) PRIO=-1
;FOLD LIN Place_R1_L2_S1_VP8 CONT Vel=0.5 m/s LPlace_R1_L2_S1_VP8 Tool[2]:Lower Gripper Base[1]:Rack1;%{PE}%R8.3.21,%MKUKATPBASIS,%CMOVE,%VLIN,%P 1:LIN, 2:Place_R1_L2_S1_VP8, 3:C_DIS C_DIS, 5:0.5, 7:LPlace_R1_L2_S1_VP8
$BWDSTART=FALSE
LDAT_ACT= LLPlace_R1_L2_S1_VP8
FDAT_ACT= FPlace_R1_L2_S1_VP8
BAS(#CP_PARAMS,0.5)
LIN XPlace_R1_L2_S1_VP8 C_DIS C_DIS
;ENDFOLD
TRIGGER WHEN DISTANCE=1 DELAY=-1 DO Schrittmerker_R1Place(10094,10093,FPlace_R1_L2_S1_VP9,XPlace_R1_L2_S1_VP9) PRIO=-1
;FOLD LIN Place_R1_L2_S1_VP9 CONT Vel=0.5 m/s LPlace_R1_L2_S1_VP9 Tool[2]:Lower Gripper Base[1]:Rack1;%{PE}%R8.3.21,%MKUKATPBASIS,%CMOVE,%VLIN,%P 1:LIN, 2:Place_R1_L2_S1_VP9, 3:C_DIS C_DIS, 5:0.5, 7:LPlace_R1_L2_S1_VP9
$BWDSTART=FALSE
LDAT_ACT= LLPlace_R1_L2_S1_VP9
FDAT_ACT= FPlace_R1_L2_S1_VP9
BAS(#CP_PARAMS,0.5)
LIN XPlace_R1_L2_S1_VP9 C_DIS C_DIS
;ENDFOLD

;FOLD Test the way back home - part 1
CONTINUE
IF ($FLAG[M_Test_GrdstFahren1] AND NOT $FLAG[M_Test_GrdstFahren2]) THEN
  $FLAG[M_Test_GrdstFahren2]=TRUE
  UP_Rueckzug( )
  RETURN
ENDIF
;ENDFOLD

;-------------------------------
; Place part position
;-------------------------------
TRIGGER WHEN DISTANCE=1 DELAY=-1 DO Schrittmerker_R1Place(10095,10096,FPlace_R1_L2_S1_AP,XPlace_R1_L2_S1_AP) PRIO=-1
;FOLD LIN Place_R1_L2_S1_AP Vel=0.2 m/s LPlace_R1_L2_S1_AP Tool[2]:Lower Gripper Base[1]:Rack1;%{PE}%R8.3.21,%MKUKATPBASIS,%CMOVE,%VLIN,%P 1:LIN, 2:Place_R1_L2_S1_AP, 3:, 5:0.2, 7:LPlace_R1_L2_S1_AP
$BWDSTART=FALSE
LDAT_ACT= LLPlace_R1_L2_S1_AP
FDAT_ACT= FPlace_R1_L2_S1_AP
BAS(#CP_PARAMS,0.2)
LIN XPlace_R1_L2_S1_AP
;ENDFOLD

;FOLD Test the way back home - part 2
CONTINUE
IF $FLAG[M_Test_GrdstFahren2] THEN
  $FLAG[M_Test_GrdstFahren2]=FALSE
  UP_Rueckzug( )
  RETURN
ENDIF
;ENDFOLD

;***************************************************
; Disable part lost detection
SetPartLostDetection(NO_PART)
;***************************************************

TRIGGER WHEN DISTANCE=1 DELAY=-1 DO Schrittmerker_R1Place(10096,10097,FPlace_R1_L2_S1_NP1,XPlace_R1_L2_S1_NP1) PRIO=-1
;FOLD LIN Place_R1_L2_S1_NP1 Vel=0.2 m/s LPlace_R1_L2_S1_NP1 Tool[2]:Lower Gripper Base[1]:Rack1;%{PE}%R8.3.21,%MKUKATPBASIS,%CMOVE,%VLIN,%P 1:LIN, 2:Place_R1_L2_S1_NP1, 3:C_DIS C_DIS, 5:0.2, 7:LPlace_R1_L2_S1_NP1
$BWDSTART=FALSE
LDAT_ACT= LLPlace_R1_L2_S1_NP1
FDAT_ACT= FPlace_R1_L2_S1_NP1
BAS(#CP_PARAMS,0.2)
LIN XPlace_R1_L2_S1_NP1
;ENDFOLD

;***************************************************
; Check for part present (empty gripper)
CheckPartPresent(EMPTY_GRIPPER)
;***************************************************
; set load data
SetLoadData( )
;***************************************************

TRIGGER WHEN DISTANCE=1 DELAY=-1 DO Schrittmerker_R1Place(10097,10098,FPlace_R1_L2_S1_NP2,XPlace_R1_L2_S1_NP2) PRIO=-1
;FOLD LIN Place_R1_L2_S1_NP2 CONT Vel=0.5 m/s LPlace_R1_L2_S1_NP2 Tool[2]:Lower Gripper Base[1]:Rack1;%{PE}%R8.3.21,%MKUKATPBASIS,%CMOVE,%VLIN,%P 1:LIN, 2:Place_R1_L2_S1_NP2, 3:C_DIS C_DIS, 5:0.5, 7:LPlace_R1_L2_S1_NP2
$BWDSTART=FALSE
LDAT_ACT= LLPlace_R1_L2_S1_NP2
FDAT_ACT= FPlace_R1_L2_S1_NP2
BAS(#CP_PARAMS,0.5)
LIN XPlace_R1_L2_S1_NP2 C_DIS C_DIS
;ENDFOLD
TRIGGER WHEN DISTANCE=1 DELAY=-1 DO Schrittmerker_R1Place(10098,10099,FPlace_R1_L2_S1_NP3,XPlace_R1_L2_S1_NP3) PRIO=-1
;FOLD LIN Place_R1_L2_S1_NP3 CONT Vel=0.5 m/s LPlace_R1_L2_S1_NP3 Tool[2]:Lower Gripper Base[1]:Rack1;%{PE}%R8.3.21,%MKUKATPBASIS,%CMOVE,%VLIN,%P 1:LIN, 2:Place_R1_L2_S1_NP3, 3:C_DIS C_DIS, 5:0.5, 7:LPlace_R1_L2_S1_NP3
$BWDSTART=FALSE
LDAT_ACT= LLPlace_R1_L2_S1_NP3
FDAT_ACT= FPlace_R1_L2_S1_NP3
BAS(#CP_PARAMS,0.5)
LIN XPlace_R1_L2_S1_NP3 C_DIS C_DIS
;ENDFOLD
TRIGGER WHEN DISTANCE=1 DELAY=-1 DO Schrittmerker_R1Place(10099,10100,FPlace_R1_L2_S1_NP4,XPlace_R1_L2_S1_NP4) PRIO=-1
;FOLD LIN Place_R1_L2_S1_NP4 Vel=0.5 m/s LPlace_R1_L2_S1_NP4 Tool[2]:Lower Gripper Base[1]:Rack1;%{PE}%R8.3.21,%MKUKATPBASIS,%CMOVE,%VLIN,%P 1:LIN, 2:Place_R1_L2_S1_NP4, 3:, 5:0.5, 7:LPlace_R1_L2_S1_NP4
$BWDSTART=FALSE
LDAT_ACT= LLPlace_R1_L2_S1_NP4
FDAT_ACT= FPlace_R1_L2_S1_NP4
BAS(#CP_PARAMS,0.5)
LIN XPlace_R1_L2_S1_NP4
;ENDFOLD
TRIGGER WHEN DISTANCE=1 DELAY=-1 DO Schrittmerker_R1Place(10100,10101,FPlace_R1_L2_S1_NP5,XPlace_R1_L2_S1_NP5) PRIO=-1
;FOLD PTP Place_R1_L2_S1_NP5 CONT Vel=100 % PPlace_R1_L2_S1_NP5 Tool[2]:Lower Gripper Base[1]:Rack1;%{PE}%R8.3.21,%MKUKATPBASIS,%CMOVE,%VPTP,%P 1:PTP, 2:Place_R1_L2_S1_NP5, 3:C_DIS, 5:100, 7:PPlace_R1_L2_S1_NP5
$BWDSTART=FALSE
PDAT_ACT= PPPlace_R1_L2_S1_NP5
FDAT_ACT= FPlace_R1_L2_S1_NP5
BAS(#PTP_PARAMS,100)
PTP XPlace_R1_L2_S1_NP5 C_DIS
;ENDFOLD
TRIGGER WHEN DISTANCE=1 DELAY=-1 DO Schrittmerker_R1Place(10101,10102,FPlace_R1_L2_S1_NP6,XPlace_R1_L2_S1_NP6) PRIO=-1
;FOLD PTP Place_R1_L2_S1_NP6 CONT Vel=100 % PPlace_R1_L2_S1_NP6 Tool[2]:Lower Gripper Base[0];%{PE}%R8.3.21,%MKUKATPBASIS,%CMOVE,%VPTP,%P 1:PTP, 2:Place_R1_L2_S1_NP6, 3:C_DIS, 5:100, 7:PPlace_R1_L2_S1_NP6
$BWDSTART=FALSE
PDAT_ACT= PPPlace_R1_L2_S1_NP6
FDAT_ACT= FPlace_R1_L2_S1_NP6
BAS(#PTP_PARAMS,100)
PTP XPlace_R1_L2_S1_NP6 C_DIS
;ENDFOLD
TRIGGER WHEN DISTANCE=1 DELAY=-1 DO Schrittmerker_R1Place(10102,10103,FPlace_R1_L2_S1_NP7,XPlace_R1_L2_S1_NP7) PRIO=-1
;FOLD PTP Place_R1_L2_S1_NP7 CONT Vel=100 % PPlace_R1_L2_S1_NP7 Tool[2]:Lower Gripper Base[0];%{PE}%R8.3.21,%MKUKATPBASIS,%CMOVE,%VPTP,%P 1:PTP, 2:Place_R1_L2_S1_NP7, 3:C_DIS, 5:100, 7:PPlace_R1_L2_S1_NP7
$BWDSTART=FALSE
PDAT_ACT= PPPlace_R1_L2_S1_NP7
FDAT_ACT= FPlace_R1_L2_S1_NP7
BAS(#PTP_PARAMS,100)
PTP XPlace_R1_L2_S1_NP7 C_DIS
;ENDFOLD
TRIGGER WHEN DISTANCE=1 DELAY=-1 DO Schrittmerker_R1Place(10103,10104,FPlace_R1_L2_S1_NP8,XPlace_R1_L2_S1_NP8) PRIO=-1
;FOLD PTP Place_R1_L2_S1_NP8 CONT Vel=100 % PPlace_R1_L2_S1_NP8 Tool[2]:Lower Gripper Base[0];%{PE}%R8.3.21,%MKUKATPBASIS,%CMOVE,%VPTP,%P 1:PTP, 2:Place_R1_L2_S1_NP8, 3:C_DIS, 5:100, 7:PPlace_R1_L2_S1_NP8
$BWDSTART=FALSE
PDAT_ACT= PPPlace_R1_L2_S1_NP8
FDAT_ACT= FPlace_R1_L2_S1_NP8
BAS(#PTP_PARAMS,100)
PTP XPlace_R1_L2_S1_NP8 C_DIS
;ENDFOLD
TRIGGER WHEN DISTANCE=1 DELAY=-1 DO Schrittmerker_R1Place(10104,10105,FPlace_R1_L2_S1_NP9,XPlace_R1_L2_S1_NP9) PRIO=-1
;FOLD PTP Place_R1_L2_S1_NP9 CONT Vel=100 % PPlace_R1_L2_S1_NP9 Tool[2]:Lower Gripper Base[0];%{PE}%R8.3.21,%MKUKATPBASIS,%CMOVE,%VPTP,%P 1:PTP, 2:Place_R1_L2_S1_NP9, 3:C_DIS, 5:100, 7:PPlace_R1_L2_S1_NP9
$BWDSTART=FALSE
PDAT_ACT= PPPlace_R1_L2_S1_NP9
FDAT_ACT= FPlace_R1_L2_S1_NP9
BAS(#PTP_PARAMS,100)
PTP XPlace_R1_L2_S1_NP9 C_DIS
;ENDFOLD

TRIGGER WHEN DISTANCE=1 DELAY=-1 DO Schrittmerker_R1Place(10105,10002,FHOME1,$nullframe,XHOME1) PRIO=-1
;FOLD PTP HOME1 Vel=100 % PHome1;%{PE}%R8.3.21,%MKUKATPBASIS,%CMOVE,%VPTP,%P 1:PTP, 2:HOME1, 3:, 5:100, 7:PHome1
$BWDSTART=FALSE
PDAT_ACT= PPHome1
FDAT_ACT= FHOME1
BAS(#PTP_PARAMS,100)
PTP XHOME1
;ENDFOLD

;***************************************************
;FOLD Final tasks.
; Robot out of area Rack 1 Level 2
RobAusStorage1_2_A68=RESET_IN_AREA
;***************************************************
; stop cyclic clearence check
$CYCFLAG[ciFreigabeSPS]=DISABLE_MONITORING
;***************************************************
; Disable collision detection
;FOLD COLLDETECT Off ;%{PE}
;FOLD Parameters ;%{h}
;Params IlfProvider=kukaroboter.basistech.inlineforms.colldetect.off; CollDetect.Command=Off
;ENDFOLD
USE_CD_PARAMS(0)
;ENDFOLD
;***************************************************
;ENDFOLD
;***************************************************

END

; ##################################################

GLOBAL DEF UP_Place_R1_L2_S2( )
;***************************************************
; Place part on:
;    Rack  1
;    Level 2
;    Shelf 2
;***************************************************
;FOLD Preconditions - Vorraussetzungen
;***************************************************
; Enable collision detection
;FOLD COLLDETECT SetLimits Axis1: 150 % Axis2: 200 % Axis3: 150 % Axis4: 200 % Axis5: 150 % Axis6: 150 % ;%{PE}
;FOLD Parameters ;%{h}
;Params IlfProvider=kukaroboter.basistech.inlineforms.colldetect.setlimits; CollDetect.Command=SetLimits; CollDetect.Axis1=150; CollDetect.Axis2=200; CollDetect.Axis3=150; CollDetect.Axis4=200; CollDetect.Axis5=150; CollDetect.Axis6=150
;ENDFOLD
SET_TQ_VALUES(150, 200, 150, 200, 150, 150)
;ENDFOLD
;***************************************************
; Check for part in gripper (tool 2).
CheckPartPresent(OCCUPIED_GRIPPER,PART_ON_TOOL_2)
;***************************************************
; Enable part lost detection for tool 2
SetPartLostDetection(PART_ON_TOOL_2)
;***************************************************
; Set load data.
SetLoadData( )
;***************************************************
; Robot has to start from home position.
IF NOT $IN_HOME1 THEN
  UP_HomeToHome(1)
ENDIF
;***************************************************
;ENDFOLD

TRIGGER WHEN DISTANCE=1 DELAY=-1 DO Schrittmerker_R1Place(10002,10002,FHOME1,$nullframe,XHOME1) PRIO=-1
;FOLD PTP HOME1 Vel=12 % PHome1;%{PE}%R8.3.21,%MKUKATPBASIS,%CMOVE,%VPTP,%P 1:PTP, 2:HOME1, 3:, 5:12, 7:PHome1
$BWDSTART=FALSE
PDAT_ACT= PPHome1
FDAT_ACT= FHOME1
BAS(#PTP_PARAMS,12)
PTP XHOME1
;ENDFOLD

;***************************************************
;FOLD Area clearence handshake.
IF NOT $FLAG[M_Inbetriebnahme] THEN
  ;-------------------------------------------------
  ; Request area clearence.
  AnfStoer_Store1_2_A100=SET_REQUEST
  ;-------------------------------------------------
  ; Wait for area clearence from PLC.
  WAIT_FOR_INPUT("Frg_Storage1_2_E68",TRUE)
  ;-------------------------------------------------
  ; Reset area clearence request.
  AnfStoer_Store1_2_A100=RESET_REQUEST
  ;-------------------------------------------------
  ; start cyclic clearence check
  $CYCFLAG[ciFreigabeSPS]=Frg_Storage1_2_E68
  ;-------------------------------------------------
ENDIF
;***************************************************
; set "robot in area"
RobAusStorage1_2_A68=SET_IN_AREA
;ENDFOLD
;***************************************************

;***************************************************
;FOLD Check for Teachmode
IF $FLAG[M_Teachen] THEN
  WAIT FOR $T1
ENDIF
;ENDFOLD
;***************************************************

; move to the rack
TRIGGER WHEN DISTANCE=1 DELAY=-1 DO Schrittmerker_R1Place(10110,10002,FPlace_R1_L2_S2_VP1,XPlace_R1_L2_S2_VP1) PRIO=-1
;FOLD PTP Place_R1_L2_S2_VP1 CONT Vel=12 % PPlace_R1_L2_S2_VP1 Tool[2]:Lower Gripper Base[0];%{PE}%R8.3.21,%MKUKATPBASIS,%CMOVE,%VPTP,%P 1:PTP, 2:Place_R1_L2_S2_VP1, 3:C_DIS, 5:12, 7:PPlace_R1_L2_S2_VP1
$BWDSTART=FALSE
PDAT_ACT= PPPlace_R1_L2_S2_VP1
FDAT_ACT= FPlace_R1_L2_S2_VP1
BAS(#PTP_PARAMS,12)
PTP XPlace_R1_L2_S2_VP1 C_DIS
;ENDFOLD
TRIGGER WHEN DISTANCE=1 DELAY=-1 DO Schrittmerker_R1Place(10111,10110,FPlace_R1_L2_S2_VP2,XPlace_R1_L2_S2_VP2) PRIO=-1
;FOLD PTP Place_R1_L2_S2_VP2 CONT Vel=12 % PPlace_R1_L2_S2_VP2 Tool[2]:Lower Gripper Base[0];%{PE}%R8.3.21,%MKUKATPBASIS,%CMOVE,%VPTP,%P 1:PTP, 2:Place_R1_L2_S2_VP2, 3:C_DIS, 5:12, 7:PPlace_R1_L2_S2_VP2
$BWDSTART=FALSE
PDAT_ACT= PPPlace_R1_L2_S2_VP2
FDAT_ACT= FPlace_R1_L2_S2_VP2
BAS(#PTP_PARAMS,12)
PTP XPlace_R1_L2_S2_VP2 C_DIS
;ENDFOLD
TRIGGER WHEN DISTANCE=1 DELAY=-1 DO Schrittmerker_R1Place(10112,10111,FPlace_R1_L2_S2_VP3,XPlace_R1_L2_S2_VP3) PRIO=-1
;FOLD PTP Place_R1_L2_S2_VP3 CONT Vel=12 % PPlace_R1_L2_S2_VP3 Tool[2]:Lower Gripper Base[0];%{PE}%R8.3.21,%MKUKATPBASIS,%CMOVE,%VPTP,%P 1:PTP, 2:Place_R1_L2_S2_VP3, 3:C_DIS, 5:12, 7:PPlace_R1_L2_S2_VP3
$BWDSTART=FALSE
PDAT_ACT= PPPlace_R1_L2_S2_VP3
FDAT_ACT= FPlace_R1_L2_S2_VP3
BAS(#PTP_PARAMS,12)
PTP XPlace_R1_L2_S2_VP3 C_DIS
;ENDFOLD
TRIGGER WHEN DISTANCE=1 DELAY=-1 DO Schrittmerker_R1Place(10113,10112,FPlace_R1_L2_S2_VP4,XPlace_R1_L2_S2_VP4) PRIO=-1
;FOLD PTP Place_R1_L2_S2_VP4 CONT Vel=12 % PPlace_R1_L2_S2_VP4 Tool[2]:Lower Gripper Base[0];%{PE}%R8.3.21,%MKUKATPBASIS,%CMOVE,%VPTP,%P 1:PTP, 2:Place_R1_L2_S2_VP4, 3:C_DIS, 5:12, 7:PPlace_R1_L2_S2_VP4
$BWDSTART=FALSE
PDAT_ACT= PPPlace_R1_L2_S2_VP4
FDAT_ACT= FPlace_R1_L2_S2_VP4
BAS(#PTP_PARAMS,12)
PTP XPlace_R1_L2_S2_VP4 C_DIS
;ENDFOLD
TRIGGER WHEN DISTANCE=1 DELAY=-1 DO Schrittmerker_R1Place(10114,10113,FPlace_R1_L2_S2_VP5,XPlace_R1_L2_S2_VP5) PRIO=-1
;FOLD PTP Place_R1_L2_S2_VP5 CONT Vel=12 % PPlace_R1_L2_S2_VP5 Tool[2]:Lower Gripper Base[0];%{PE}%R8.3.21,%MKUKATPBASIS,%CMOVE,%VPTP,%P 1:PTP, 2:Place_R1_L2_S2_VP5, 3:C_DIS, 5:12, 7:PPlace_R1_L2_S2_VP5
$BWDSTART=FALSE
PDAT_ACT= PPPlace_R1_L2_S2_VP5
FDAT_ACT= FPlace_R1_L2_S2_VP5
BAS(#PTP_PARAMS,12)
PTP XPlace_R1_L2_S2_VP5 C_DIS
;ENDFOLD
TRIGGER WHEN DISTANCE=1 DELAY=-1 DO Schrittmerker_R1Place(10115,10114,FPlace_R1_L2_S2_VP6,XPlace_R1_L2_S2_VP6) PRIO=-1
;FOLD PTP Place_R1_L2_S2_VP6 CONT Vel=12 % PPlace_R1_L2_S2_VP6 Tool[2]:Lower Gripper Base[1]:Rack1;%{PE}%R8.3.21,%MKUKATPBASIS,%CMOVE,%VPTP,%P 1:PTP, 2:Place_R1_L2_S2_VP6, 3:C_DIS, 5:12, 7:PPlace_R1_L2_S2_VP6
$BWDSTART=FALSE
PDAT_ACT= PPPlace_R1_L2_S2_VP6
FDAT_ACT= FPlace_R1_L2_S2_VP6
BAS(#PTP_PARAMS,12)
PTP XPlace_R1_L2_S2_VP6 C_DIS
;ENDFOLD
TRIGGER WHEN DISTANCE=1 DELAY=-1 DO Schrittmerker_R1Place(10116,10115,FPlace_R1_L2_S2_VP7,XPlace_R1_L2_S2_VP7) PRIO=-1
;FOLD PTP Place_R1_L2_S2_VP7 CONT Vel=12 % PPlace_R1_L2_S2_VP7 Tool[2]:Lower Gripper Base[1]:Rack1;%{PE}%R8.3.21,%MKUKATPBASIS,%CMOVE,%VPTP,%P 1:PTP, 2:Place_R1_L2_S2_VP7, 3:C_DIS, 5:12, 7:PPlace_R1_L2_S2_VP7
$BWDSTART=FALSE
PDAT_ACT= PPPlace_R1_L2_S2_VP7
FDAT_ACT= FPlace_R1_L2_S2_VP7
BAS(#PTP_PARAMS,12)
PTP XPlace_R1_L2_S2_VP7 C_DIS
;ENDFOLD

TRIGGER WHEN DISTANCE=1 DELAY=-1 DO Schrittmerker_R1Place(10117,10116,FPlace_R1_L2_S2_Check,XPlace_R1_L2_S2_Check) PRIO=-1
;FOLD PTP Place_R1_L2_S2_Check Vel=12 % PPlace_R1_L2_S2_Check Tool[2]:Lower Gripper Base[1]:Rack1;%{PE}%R8.3.21,%MKUKATPBASIS,%CMOVE,%VPTP,%P 1:PTP, 2:Place_R1_L2_S2_Check, 3:, 5:12, 7:PPlace_R1_L2_S2_Check
$BWDSTART=FALSE
PDAT_ACT= PPPlace_R1_L2_S2_Check
FDAT_ACT= FPlace_R1_L2_S2_Check
BAS(#PTP_PARAMS,12)
PTP XPlace_R1_L2_S2_Check
;ENDFOLD

;***************************************************
;FOLD Pruefe Platz frei
IF (DetectPart(CHECK_SHELF,PLACE)==OCCUPIED) THEN
  UP_Rueckzug_R1Place( )
  RETURN
ENDIF
;ENDFOLD
;***************************************************

TRIGGER WHEN DISTANCE=1 DELAY=-1 DO Schrittmerker_R1Place(10118,10117,FPlace_R1_L2_S2_VP8,XPlace_R1_L2_S2_VP8) PRIO=-1
;FOLD LIN Place_R1_L2_S2_VP8 CONT Vel=0.5 m/s LPlace_R1_L2_S2_VP8 Tool[2]:Lower Gripper Base[1]:Rack1;%{PE}%R8.3.21,%MKUKATPBASIS,%CMOVE,%VLIN,%P 1:LIN, 2:Place_R1_L2_S2_VP8, 3:C_DIS C_DIS, 5:0.5, 7:LPlace_R1_L2_S2_VP8
$BWDSTART=FALSE
LDAT_ACT= LLPlace_R1_L2_S2_VP8
FDAT_ACT= FPlace_R1_L2_S2_VP8
BAS(#CP_PARAMS,0.5)
LIN XPlace_R1_L2_S2_VP8 C_DIS C_DIS
;ENDFOLD
TRIGGER WHEN DISTANCE=1 DELAY=-1 DO Schrittmerker_R1Place(10119,10118,FPlace_R1_L2_S2_VP9,XPlace_R1_L2_S2_VP9) PRIO=-1
;FOLD LIN Place_R1_L2_S2_VP9 CONT Vel=0.5 m/s LPlace_R1_L2_S2_VP9 Tool[2]:Lower Gripper Base[1]:Rack1;%{PE}%R8.3.21,%MKUKATPBASIS,%CMOVE,%VLIN,%P 1:LIN, 2:Place_R1_L2_S2_VP9, 3:C_DIS C_DIS, 5:0.5, 7:LPlace_R1_L2_S2_VP9
$BWDSTART=FALSE
LDAT_ACT= LLPlace_R1_L2_S2_VP9
FDAT_ACT= FPlace_R1_L2_S2_VP9
BAS(#CP_PARAMS,0.5)
LIN XPlace_R1_L2_S2_VP9 C_DIS C_DIS
;ENDFOLD

;FOLD Test the way back home - part 1
CONTINUE
IF ($FLAG[M_Test_GrdstFahren1] AND NOT $FLAG[M_Test_GrdstFahren2]) THEN
  $FLAG[M_Test_GrdstFahren2]=TRUE
  UP_Rueckzug( )
  RETURN
ENDIF
;ENDFOLD

;-------------------------------
; Place part position
;-------------------------------
TRIGGER WHEN DISTANCE=1 DELAY=-1 DO Schrittmerker_R1Place(10120,10121,FPlace_R1_L2_S2_AP,XPlace_R1_L2_S2_AP) PRIO=-1
;FOLD LIN Place_R1_L2_S2_AP Vel=0.2 m/s LPlace_R1_L2_S2_AP Tool[2]:Lower Gripper Base[1]:Rack1;%{PE}%R8.3.21,%MKUKATPBASIS,%CMOVE,%VLIN,%P 1:LIN, 2:Place_R1_L2_S2_AP, 3:, 5:0.2, 7:LPlace_R1_L2_S2_AP
$BWDSTART=FALSE
LDAT_ACT= LLPlace_R1_L2_S2_AP
FDAT_ACT= FPlace_R1_L2_S2_AP
BAS(#CP_PARAMS,0.2)
LIN XPlace_R1_L2_S2_AP
;ENDFOLD

;FOLD Test the way back home - part 2
CONTINUE
IF $FLAG[M_Test_GrdstFahren2] THEN
  $FLAG[M_Test_GrdstFahren2]=FALSE
  UP_Rueckzug( )
  RETURN
ENDIF
;ENDFOLD

;***************************************************
; Disable part lost detection
SetPartLostDetection(NO_PART)
;***************************************************

TRIGGER WHEN DISTANCE=1 DELAY=-1 DO Schrittmerker_R1Place(10121,10122,FPlace_R1_L2_S2_NP1,XPlace_R1_L2_S2_NP1) PRIO=-1
;FOLD LIN Place_R1_L2_S2_NP1 Vel=0.2 m/s LPlace_R1_L2_S2_NP1 Tool[2]:Lower Gripper Base[1]:Rack1;%{PE}%R8.3.21,%MKUKATPBASIS,%CMOVE,%VLIN,%P 1:LIN, 2:Place_R1_L2_S2_NP1, 3:C_DIS C_DIS, 5:0.2, 7:LPlace_R1_L2_S2_NP1
$BWDSTART=FALSE
LDAT_ACT= LLPlace_R1_L2_S2_NP1
FDAT_ACT= FPlace_R1_L2_S2_NP1
BAS(#CP_PARAMS,0.2)
LIN XPlace_R1_L2_S2_NP1
;ENDFOLD

;***************************************************
; Check for part present (empty gripper)
CheckPartPresent(EMPTY_GRIPPER)
;***************************************************
; set load data
SetLoadData( )
;***************************************************

TRIGGER WHEN DISTANCE=1 DELAY=-1 DO Schrittmerker_R1Place(10122,10123,FPlace_R1_L2_S2_NP2,XPlace_R1_L2_S2_NP2) PRIO=-1
;FOLD LIN Place_R1_L2_S2_NP2 CONT Vel=0.5 m/s LPlace_R1_L2_S2_NP2 Tool[2]:Lower Gripper Base[1]:Rack1;%{PE}%R8.3.21,%MKUKATPBASIS,%CMOVE,%VLIN,%P 1:LIN, 2:Place_R1_L2_S2_NP2, 3:C_DIS C_DIS, 5:0.5, 7:LPlace_R1_L2_S2_NP2
$BWDSTART=FALSE
LDAT_ACT= LLPlace_R1_L2_S2_NP2
FDAT_ACT= FPlace_R1_L2_S2_NP2
BAS(#CP_PARAMS,0.5)
LIN XPlace_R1_L2_S2_NP2 C_DIS C_DIS
;ENDFOLD
TRIGGER WHEN DISTANCE=1 DELAY=-1 DO Schrittmerker_R1Place(10123,10124,FPlace_R1_L2_S2_NP3,XPlace_R1_L2_S2_NP3) PRIO=-1
;FOLD LIN Place_R1_L2_S2_NP3 Vel=0.5 m/s LPlace_R1_L2_S2_NP3 Tool[2]:Lower Gripper Base[1]:Rack 1 ;%{PE}
$BWDSTART=FALSE
LDAT_ACT=LLPlace_R1_L2_S2_NP3
FDAT_ACT=FPlace_R1_L2_S2_NP3
BAS(#CP_PARAMS, 0.5)
LIN XPlace_R1_L2_S2_NP3
;ENDFOLD
TRIGGER WHEN DISTANCE=1 DELAY=-1 DO Schrittmerker_R1Place(10124,10125,FPlace_R1_L2_S2_NP4,XPlace_R1_L2_S2_NP4) PRIO=-1
;FOLD PTP Place_R1_L2_S2_NP4 CONT Vel=100 % PPlace_R1_L2_S2_NP4 Tool[2]:Lower Gripper Base[0];%{PE}%R8.3.21,%MKUKATPBASIS,%CMOVE,%VPTP,%P 1:PTP, 2:Place_R1_L2_S2_NP4, 3:C_DIS, 5:100, 7:PPlace_R1_L2_S2_NP4
$BWDSTART=FALSE
PDAT_ACT= PPPlace_R1_L2_S2_NP4
FDAT_ACT= FPlace_R1_L2_S2_NP4
BAS(#PTP_PARAMS,100)
PTP XPlace_R1_L2_S2_NP4 C_DIS
;ENDFOLD
TRIGGER WHEN DISTANCE=1 DELAY=-1 DO Schrittmerker_R1Place(10125,10126,FPlace_R1_L2_S2_NP5,XPlace_R1_L2_S2_NP5) PRIO=-1
;FOLD PTP Place_R1_L2_S2_NP5 CONT Vel=100 % PPlace_R1_L2_S2_NP5 Tool[2]:Lower Gripper Base[0];%{PE}%R8.3.21,%MKUKATPBASIS,%CMOVE,%VPTP,%P 1:PTP, 2:Place_R1_L2_S2_NP5, 3:C_DIS, 5:100, 7:PPlace_R1_L2_S2_NP5
$BWDSTART=FALSE
PDAT_ACT= PPPlace_R1_L2_S2_NP5
FDAT_ACT= FPlace_R1_L2_S2_NP5
BAS(#PTP_PARAMS,100)
PTP XPlace_R1_L2_S2_NP5 C_DIS
;ENDFOLD
TRIGGER WHEN DISTANCE=1 DELAY=-1 DO Schrittmerker_R1Place(10126,10127,FPlace_R1_L2_S2_NP6,XPlace_R1_L2_S2_NP6) PRIO=-1
;FOLD PTP Place_R1_L2_S2_NP6 CONT Vel=100 % PPlace_R1_L2_S2_NP6 Tool[2]:Lower Gripper Base[0];%{PE}%R8.3.21,%MKUKATPBASIS,%CMOVE,%VPTP,%P 1:PTP, 2:Place_R1_L2_S2_NP6, 3:C_DIS, 5:100, 7:PPlace_R1_L2_S2_NP6
$BWDSTART=FALSE
PDAT_ACT= PPPlace_R1_L2_S2_NP6
FDAT_ACT= FPlace_R1_L2_S2_NP6
BAS(#PTP_PARAMS,100)
PTP XPlace_R1_L2_S2_NP6 C_DIS
;ENDFOLD
TRIGGER WHEN DISTANCE=1 DELAY=-1 DO Schrittmerker_R1Place(10127,10128,FPlace_R1_L2_S2_NP7,XPlace_R1_L2_S2_NP7) PRIO=-1
;FOLD PTP Place_R1_L2_S2_NP7 CONT Vel=100 % PPlace_R1_L2_S2_NP7 Tool[2]:Lower Gripper Base[0];%{PE}%R8.3.21,%MKUKATPBASIS,%CMOVE,%VPTP,%P 1:PTP, 2:Place_R1_L2_S2_NP7, 3:C_DIS, 5:100, 7:PPlace_R1_L2_S2_NP7
$BWDSTART=FALSE
PDAT_ACT= PPPlace_R1_L2_S2_NP7
FDAT_ACT= FPlace_R1_L2_S2_NP7
BAS(#PTP_PARAMS,100)
PTP XPlace_R1_L2_S2_NP7 C_DIS
;ENDFOLD

TRIGGER WHEN DISTANCE=1 DELAY=-1 DO Schrittmerker_R1Place(10128,10002,FHOME1,$nullframe,XHOME1) PRIO=-1
;FOLD PTP HOME1 Vel=100 % PHome1;%{PE}%R8.3.21,%MKUKATPBASIS,%CMOVE,%VPTP,%P 1:PTP, 2:HOME1, 3:, 5:100, 7:PHome1
$BWDSTART=FALSE
PDAT_ACT= PPHome1
FDAT_ACT= FHOME1
BAS(#PTP_PARAMS,100)
PTP XHOME1
;ENDFOLD

;***************************************************
;FOLD Final tasks.
; Robot out of area Rack 1 Level 2
RobAusStorage1_2_A68=RESET_IN_AREA
;***************************************************
; stop cyclic clearence check
$CYCFLAG[ciFreigabeSPS]=DISABLE_MONITORING
;***************************************************
; Disable collision detection
;FOLD COLLDETECT Off ;%{PE}
;FOLD Parameters ;%{h}
;Params IlfProvider=kukaroboter.basistech.inlineforms.colldetect.off; CollDetect.Command=Off
;ENDFOLD
USE_CD_PARAMS(0)
;ENDFOLD
;***************************************************
;ENDFOLD
;***************************************************

END

; ##################################################

GLOBAL DEF UP_Place_R1_L2_S3( )
;***************************************************
; Place part on:
;    Rack  1
;    Level 2
;    Shelf 3
;***************************************************
;FOLD Preconditions - Vorraussetzungen
;***************************************************
; Enable collision detection
;FOLD COLLDETECT SetLimits Axis1: 150 % Axis2: 200 % Axis3: 150 % Axis4: 200 % Axis5: 150 % Axis6: 150 % ;%{PE}
;FOLD Parameters ;%{h}
;Params IlfProvider=kukaroboter.basistech.inlineforms.colldetect.setlimits; CollDetect.Command=SetLimits; CollDetect.Axis1=150; CollDetect.Axis2=200; CollDetect.Axis3=150; CollDetect.Axis4=200; CollDetect.Axis5=150; CollDetect.Axis6=150
;ENDFOLD
SET_TQ_VALUES(150, 200, 150, 200, 150, 150)
;ENDFOLD
;***************************************************
; Check for part in gripper (tool 2).
CheckPartPresent(OCCUPIED_GRIPPER,PART_ON_TOOL_2)
;***************************************************
; Enable part lost detection for tool 2
SetPartLostDetection(PART_ON_TOOL_2)
;***************************************************
; Set load data.
SetLoadData( )
;***************************************************
; Robot has to start from home position.
IF NOT $IN_HOME1 THEN
  UP_HomeToHome(1)
ENDIF
;***************************************************
;ENDFOLD

TRIGGER WHEN DISTANCE=1 DELAY=-1 DO Schrittmerker_R1Place(10002,10002,FHOME1,$nullframe,XHOME1) PRIO=-1
;FOLD PTP HOME1 Vel=12 % PHome1;%{PE}%R8.3.21,%MKUKATPBASIS,%CMOVE,%VPTP,%P 1:PTP, 2:HOME1, 3:, 5:12, 7:PHome1
$BWDSTART=FALSE
PDAT_ACT= PPHome1
FDAT_ACT= FHOME1
BAS(#PTP_PARAMS,12)
PTP XHOME1
;ENDFOLD

;***************************************************
;FOLD Area clearence handshake.
IF NOT $FLAG[M_Inbetriebnahme] THEN
  ;-------------------------------------------------
  ; Request area clearence.
  AnfStoer_Store1_2_A100=SET_REQUEST
  ;-------------------------------------------------
  ; Wait for area clearence from PLC.
  WAIT_FOR_INPUT("Frg_Storage1_2_E68",TRUE)
  ;-------------------------------------------------
  ; Reset area clearence request.
  AnfStoer_Store1_2_A100=RESET_REQUEST
  ;-------------------------------------------------
  ; start cyclic clearence check
  $CYCFLAG[ciFreigabeSPS]=Frg_Storage1_2_E68
  ;-------------------------------------------------
ENDIF
;***************************************************
; set "robot in area"
RobAusStorage1_2_A68=SET_IN_AREA
;ENDFOLD
;***************************************************

;***************************************************
;FOLD Check for Teachmode
IF $FLAG[M_Teachen] THEN
  WAIT FOR $T1
ENDIF
;ENDFOLD
;***************************************************

; move to the rack
TRIGGER WHEN DISTANCE=1 DELAY=-1 DO Schrittmerker_R1Place(10130,10002,FPlace_R1_L2_S3_VP1,XPlace_R1_L2_S3_VP1) PRIO=-1
;FOLD PTP Place_R1_L2_S3_VP1 CONT Vel=12 % PPlace_R1_L2_S3_VP1 Tool[2]:Lower Gripper Base[0];%{PE}%R8.3.21,%MKUKATPBASIS,%CMOVE,%VPTP,%P 1:PTP, 2:Place_R1_L2_S3_VP1, 3:C_DIS, 5:12, 7:PPlace_R1_L2_S3_VP1
$BWDSTART=FALSE
PDAT_ACT= PPPlace_R1_L2_S3_VP1
FDAT_ACT= FPlace_R1_L2_S3_VP1
BAS(#PTP_PARAMS,12)
PTP XPlace_R1_L2_S3_VP1 C_DIS
;ENDFOLD
TRIGGER WHEN DISTANCE=1 DELAY=-1 DO Schrittmerker_R1Place(10131,10130,FPlace_R1_L2_S3_VP2,XPlace_R1_L2_S3_VP2) PRIO=-1
;FOLD PTP Place_R1_L2_S3_VP2 CONT Vel=12 % PPlace_R1_L2_S3_VP2 Tool[2]:Lower Gripper Base[0];%{PE}%R8.3.21,%MKUKATPBASIS,%CMOVE,%VPTP,%P 1:PTP, 2:Place_R1_L2_S3_VP2, 3:C_DIS, 5:12, 7:PPlace_R1_L2_S3_VP2
$BWDSTART=FALSE
PDAT_ACT= PPPlace_R1_L2_S3_VP2
FDAT_ACT= FPlace_R1_L2_S3_VP2
BAS(#PTP_PARAMS,12)
PTP XPlace_R1_L2_S3_VP2 C_DIS
;ENDFOLD
TRIGGER WHEN DISTANCE=1 DELAY=-1 DO Schrittmerker_R1Place(10132,10131,FPlace_R1_L2_S3_VP3,XPlace_R1_L2_S3_VP3) PRIO=-1
;FOLD PTP Place_R1_L2_S3_VP3 CONT Vel=12 % PPlace_R1_L2_S3_VP3 Tool[2]:Lower Gripper Base[0];%{PE}%R8.3.21,%MKUKATPBASIS,%CMOVE,%VPTP,%P 1:PTP, 2:Place_R1_L2_S3_VP3, 3:C_DIS, 5:12, 7:PPlace_R1_L2_S3_VP3
$BWDSTART=FALSE
PDAT_ACT= PPPlace_R1_L2_S3_VP3
FDAT_ACT= FPlace_R1_L2_S3_VP3
BAS(#PTP_PARAMS,12)
PTP XPlace_R1_L2_S3_VP3 C_DIS
;ENDFOLD
TRIGGER WHEN DISTANCE=1 DELAY=-1 DO Schrittmerker_R1Place(10133,10132,FPlace_R1_L2_S3_VP4,XPlace_R1_L2_S3_VP4) PRIO=-1
;FOLD PTP Place_R1_L2_S3_VP4 CONT Vel=12 % PPlace_R1_L2_S3_VP4 Tool[2]:Lower Gripper Base[0];%{PE}%R8.3.21,%MKUKATPBASIS,%CMOVE,%VPTP,%P 1:PTP, 2:Place_R1_L2_S3_VP4, 3:C_DIS, 5:12, 7:PPlace_R1_L2_S3_VP4
$BWDSTART=FALSE
PDAT_ACT= PPPlace_R1_L2_S3_VP4
FDAT_ACT= FPlace_R1_L2_S3_VP4
BAS(#PTP_PARAMS,12)
PTP XPlace_R1_L2_S3_VP4 C_DIS
;ENDFOLD
TRIGGER WHEN DISTANCE=1 DELAY=-1 DO Schrittmerker_R1Place(10134,10133,FPlace_R1_L2_S3_VP5,XPlace_R1_L2_S3_VP5) PRIO=-1
;FOLD PTP Place_R1_L2_S3_VP5 CONT Vel=12 % PPlace_R1_L2_S3_VP5 Tool[2]:Lower Gripper Base[1]:Rack1;%{PE}%R8.3.21,%MKUKATPBASIS,%CMOVE,%VPTP,%P 1:PTP, 2:Place_R1_L2_S3_VP5, 3:C_DIS, 5:12, 7:PPlace_R1_L2_S3_VP5
$BWDSTART=FALSE
PDAT_ACT= PPPlace_R1_L2_S3_VP5
FDAT_ACT= FPlace_R1_L2_S3_VP5
BAS(#PTP_PARAMS,12)
PTP XPlace_R1_L2_S3_VP5 C_DIS
;ENDFOLD

TRIGGER WHEN DISTANCE=1 DELAY=-1 DO Schrittmerker_R1Place(10135,10134,FPlace_R1_L2_S3_Check,XPlace_R1_L2_S3_Check) PRIO=-1
;FOLD PTP Place_R1_L2_S3_Check Vel=12 % PPlace_R1_L2_S3_Check Tool[2]:Lower Gripper Base[1]:Rack1;%{PE}%R8.3.21,%MKUKATPBASIS,%CMOVE,%VPTP,%P 1:PTP, 2:Place_R1_L2_S3_Check, 3:, 5:12, 7:PPlace_R1_L2_S3_Check
$BWDSTART=FALSE
PDAT_ACT= PPPlace_R1_L2_S3_Check
FDAT_ACT= FPlace_R1_L2_S3_Check
BAS(#PTP_PARAMS,12)
PTP XPlace_R1_L2_S3_Check
;ENDFOLD

;***************************************************
;FOLD Pruefe Platz frei
IF (DetectPart(CHECK_SHELF,PLACE)==OCCUPIED) THEN
  UP_Rueckzug_R1Place( )
  RETURN
ENDIF
;ENDFOLD
;***************************************************

TRIGGER WHEN DISTANCE=1 DELAY=-1 DO Schrittmerker_R1Place(10136,10135,FPlace_R1_L2_S3_VP6,XPlace_R1_L2_S3_VP6) PRIO=-1
;FOLD LIN Place_R1_L2_S3_VP6 CONT Vel=0.5 m/s LPlace_R1_L2_S3_VP6 Tool[2]:Lower Gripper Base[1]:Rack1;%{PE}%R8.3.21,%MKUKATPBASIS,%CMOVE,%VLIN,%P 1:LIN, 2:Place_R1_L2_S3_VP6, 3:C_DIS C_DIS, 5:0.5, 7:LPlace_R1_L2_S3_VP6
$BWDSTART=FALSE
LDAT_ACT= LLPlace_R1_L2_S3_VP6
FDAT_ACT= FPlace_R1_L2_S3_VP6
BAS(#CP_PARAMS,0.5)
LIN XPlace_R1_L2_S3_VP6 C_DIS C_DIS
;ENDFOLD

;FOLD Test the way back home - part 1
CONTINUE
IF ($FLAG[M_Test_GrdstFahren1] AND NOT $FLAG[M_Test_GrdstFahren2]) THEN
  $FLAG[M_Test_GrdstFahren2]=TRUE
  UP_Rueckzug( )
  RETURN
ENDIF
;ENDFOLD

;-------------------------------
; Place part position
;-------------------------------
TRIGGER WHEN DISTANCE=1 DELAY=-1 DO Schrittmerker_R1Place(10137,10138,FPlace_R1_L2_S3_AP,XPlace_R1_L2_S3_AP) PRIO=-1
;FOLD LIN Place_R1_L2_S3_AP Vel=0.2 m/s LPlace_R1_L2_S3_AP Tool[2]:Lower Gripper Base[1]:Rack1;%{PE}%R8.3.21,%MKUKATPBASIS,%CMOVE,%VLIN,%P 1:LIN, 2:Place_R1_L2_S3_AP, 3:, 5:0.2, 7:LPlace_R1_L2_S3_AP
$BWDSTART=FALSE
LDAT_ACT= LLPlace_R1_L2_S3_AP
FDAT_ACT= FPlace_R1_L2_S3_AP
BAS(#CP_PARAMS,0.2)
LIN XPlace_R1_L2_S3_AP
;ENDFOLD

;FOLD Test the way back home - part 2
CONTINUE
IF $FLAG[M_Test_GrdstFahren2] THEN
  $FLAG[M_Test_GrdstFahren2]=FALSE
  UP_Rueckzug( )
  RETURN
ENDIF
;ENDFOLD

;***************************************************
; Disable part lost detection
SetPartLostDetection(NO_PART)
;***************************************************

TRIGGER WHEN DISTANCE=1 DELAY=-1 DO Schrittmerker_R1Place(10138,10139,FPlace_R1_L2_S3_NP1,XPlace_R1_L2_S3_NP1) PRIO=-1
;FOLD LIN Place_R1_L2_S3_NP1 Vel=0.2 m/s LPlace_R1_L2_S3_NP1 Tool[2]:Lower Gripper Base[1]:Rack1;%{PE}%R8.3.21,%MKUKATPBASIS,%CMOVE,%VLIN,%P 1:LIN, 2:Place_R1_L2_S3_NP1, 3:C_DIS C_DIS, 5:0.2, 7:LPlace_R1_L2_S3_NP1
$BWDSTART=FALSE
LDAT_ACT= LLPlace_R1_L2_S3_NP1
FDAT_ACT= FPlace_R1_L2_S3_NP1
BAS(#CP_PARAMS,0.2)
LIN XPlace_R1_L2_S3_NP1
;ENDFOLD

;***************************************************
; Check for part present (empty gripper)
CheckPartPresent(EMPTY_GRIPPER)
;***************************************************
; set load data
SetLoadData( )
;***************************************************

TRIGGER WHEN DISTANCE=1 DELAY=-1 DO Schrittmerker_R1Place(10139,10140,FPlace_R1_L2_S3_NP2,XPlace_R1_L2_S3_NP2) PRIO=-1
;FOLD LIN Place_R1_L2_S3_NP2 CONT Vel=0.5 m/s LPlace_R1_L2_S3_NP2 Tool[2]:Lower Gripper Base[1]:Rack1;%{PE}%R8.3.21,%MKUKATPBASIS,%CMOVE,%VLIN,%P 1:LIN, 2:Place_R1_L2_S3_NP2, 3:C_DIS C_DIS, 5:0.5, 7:LPlace_R1_L2_S3_NP2
$BWDSTART=FALSE
LDAT_ACT= LLPlace_R1_L2_S3_NP2
FDAT_ACT= FPlace_R1_L2_S3_NP2
BAS(#CP_PARAMS,0.5)
LIN XPlace_R1_L2_S3_NP2 C_DIS C_DIS
;ENDFOLD
TRIGGER WHEN DISTANCE=1 DELAY=-1 DO Schrittmerker_R1Place(10140,10141,FPlace_R1_L2_S3_NP3,XPlace_R1_L2_S3_NP3) PRIO=-1
;FOLD LIN Place_R1_L2_S3_NP3 CONT Vel=0.5 m/s LPlace_R1_L2_S3_NP3 Tool[2]:Lower Gripper Base[1]:Rack1;%{PE}%R8.3.21,%MKUKATPBASIS,%CMOVE,%VLIN,%P 1:LIN, 2:Place_R1_L2_S3_NP3, 3:C_DIS C_DIS, 5:0.5, 7:LPlace_R1_L2_S3_NP3
$BWDSTART=FALSE
LDAT_ACT= LLPlace_R1_L2_S3_NP3
FDAT_ACT= FPlace_R1_L2_S3_NP3
BAS(#CP_PARAMS,0.5)
LIN XPlace_R1_L2_S3_NP3 C_DIS C_DIS
;ENDFOLD
TRIGGER WHEN DISTANCE=1 DELAY=-1 DO Schrittmerker_R1Place(10141,10142,FPlace_R1_L2_S3_NP4,XPlace_R1_L2_S3_NP4) PRIO=-1
;FOLD PTP Place_R1_L2_S3_NP4 CONT Vel=100 % PPlace_R1_L2_S3_NP4 Tool[2]:Lower Gripper Base[0];%{PE}%R8.3.21,%MKUKATPBASIS,%CMOVE,%VPTP,%P 1:PTP, 2:Place_R1_L2_S3_NP4, 3:C_DIS, 5:100, 7:PPlace_R1_L2_S3_NP4
$BWDSTART=FALSE
PDAT_ACT= PPPlace_R1_L2_S3_NP4
FDAT_ACT= FPlace_R1_L2_S3_NP4
BAS(#PTP_PARAMS,100)
PTP XPlace_R1_L2_S3_NP4 C_DIS
;ENDFOLD
TRIGGER WHEN DISTANCE=1 DELAY=-1 DO Schrittmerker_R1Place(10142,10143,FPlace_R1_L2_S3_NP5,XPlace_R1_L2_S3_NP5) PRIO=-1
;FOLD PTP Place_R1_L2_S3_NP5 CONT Vel=100 % PPlace_R1_L2_S3_NP5 Tool[2]:Lower Gripper Base[0];%{PE}%R8.3.21,%MKUKATPBASIS,%CMOVE,%VPTP,%P 1:PTP, 2:Place_R1_L2_S3_NP5, 3:C_DIS, 5:100, 7:PPlace_R1_L2_S3_NP5
$BWDSTART=FALSE
PDAT_ACT= PPPlace_R1_L2_S3_NP5
FDAT_ACT= FPlace_R1_L2_S3_NP5
BAS(#PTP_PARAMS,100)
PTP XPlace_R1_L2_S3_NP5 C_DIS
;ENDFOLD
TRIGGER WHEN DISTANCE=1 DELAY=-1 DO Schrittmerker_R1Place(10143,10144,FPlace_R1_L2_S3_NP6,XPlace_R1_L2_S3_NP6) PRIO=-1
;FOLD PTP Place_R1_L2_S3_NP6 CONT Vel=100 % PPlace_R1_L2_S3_NP6 Tool[2]:Lower Gripper Base[0];%{PE}%R8.3.21,%MKUKATPBASIS,%CMOVE,%VPTP,%P 1:PTP, 2:Place_R1_L2_S3_NP6, 3:C_DIS, 5:100, 7:PPlace_R1_L2_S3_NP6
$BWDSTART=FALSE
PDAT_ACT= PPPlace_R1_L2_S3_NP6
FDAT_ACT= FPlace_R1_L2_S3_NP6
BAS(#PTP_PARAMS,100)
PTP XPlace_R1_L2_S3_NP6 C_DIS
;ENDFOLD
TRIGGER WHEN DISTANCE=1 DELAY=-1 DO Schrittmerker_R1Place(10144,10145,FPlace_R1_L2_S3_NP7,XPlace_R1_L2_S3_NP7) PRIO=-1
;FOLD PTP Place_R1_L2_S3_NP7 CONT Vel=100 % PPlace_R1_L2_S3_NP7 Tool[2]:Lower Gripper Base[0];%{PE}%R8.3.21,%MKUKATPBASIS,%CMOVE,%VPTP,%P 1:PTP, 2:Place_R1_L2_S3_NP7, 3:C_DIS, 5:100, 7:PPlace_R1_L2_S3_NP7
$BWDSTART=FALSE
PDAT_ACT= PPPlace_R1_L2_S3_NP7
FDAT_ACT= FPlace_R1_L2_S3_NP7
BAS(#PTP_PARAMS,100)
PTP XPlace_R1_L2_S3_NP7 C_DIS
;ENDFOLD

TRIGGER WHEN DISTANCE=1 DELAY=-1 DO Schrittmerker_R1Place(10145,10002,FHOME1,$nullframe,XHOME1) PRIO=-1
;FOLD PTP HOME1 Vel=100 % PHome1;%{PE}%R8.3.21,%MKUKATPBASIS,%CMOVE,%VPTP,%P 1:PTP, 2:HOME1, 3:, 5:100, 7:PHome1
$BWDSTART=FALSE
PDAT_ACT= PPHome1
FDAT_ACT= FHOME1
BAS(#PTP_PARAMS,100)
PTP XHOME1
;ENDFOLD

;***************************************************
;FOLD Final tasks.
; Robot out of area Rack 1 Level 2
RobAusStorage1_2_A68=RESET_IN_AREA
;***************************************************
; stop cyclic clearence check
$CYCFLAG[ciFreigabeSPS]=DISABLE_MONITORING
;***************************************************
; Disable collision detection
;FOLD COLLDETECT Off ;%{PE}
;FOLD Parameters ;%{h}
;Params IlfProvider=kukaroboter.basistech.inlineforms.colldetect.off; CollDetect.Command=Off
;ENDFOLD
USE_CD_PARAMS(0)
;ENDFOLD
;***************************************************
;ENDFOLD
;***************************************************

END

; ##################################################

GLOBAL DEF UP_Place_R1_L2_S4( )
;***************************************************
; Place part on:
;    Rack  1
;    Level 2
;    Shelf 4
;***************************************************
;FOLD Preconditions - Vorraussetzungen
;***************************************************
; Enable collision detection
;FOLD COLLDETECT SetLimits Axis1: 150 % Axis2: 200 % Axis3: 150 % Axis4: 200 % Axis5: 150 % Axis6: 150 % ;%{PE}
;FOLD Parameters ;%{h}
;Params IlfProvider=kukaroboter.basistech.inlineforms.colldetect.setlimits; CollDetect.Command=SetLimits; CollDetect.Axis1=150; CollDetect.Axis2=200; CollDetect.Axis3=150; CollDetect.Axis4=200; CollDetect.Axis5=150; CollDetect.Axis6=150
;ENDFOLD
SET_TQ_VALUES(150, 200, 150, 200, 150, 150)
;ENDFOLD
;***************************************************
; Check for part in gripper (tool 2).
CheckPartPresent(OCCUPIED_GRIPPER,PART_ON_TOOL_2)
;***************************************************
; Enable part lost detection for tool 2
SetPartLostDetection(PART_ON_TOOL_2)
;***************************************************
; Set load data.
SetLoadData( )
;***************************************************
; Robot has to start from home position.
IF NOT $IN_HOME1 THEN
  UP_HomeToHome(1)
ENDIF
;***************************************************
;ENDFOLD

TRIGGER WHEN DISTANCE=1 DELAY=-1 DO Schrittmerker_R1Place(10002,10002,FHOME1,$nullframe,XHOME1) PRIO=-1
;FOLD PTP HOME1 Vel=12 % PHome1;%{PE}%R8.3.21,%MKUKATPBASIS,%CMOVE,%VPTP,%P 1:PTP, 2:HOME1, 3:, 5:12, 7:PHome1
$BWDSTART=FALSE
PDAT_ACT= PPHome1
FDAT_ACT= FHOME1
BAS(#PTP_PARAMS,12)
PTP XHOME1
;ENDFOLD

;***************************************************
;FOLD Area clearence handshake.
IF NOT $FLAG[M_Inbetriebnahme] THEN
  ;-------------------------------------------------
  ; Request area clearence.
  AnfStoer_Store1_2_A100=SET_REQUEST
  ;-------------------------------------------------
  ; Wait for area clearence from PLC.
  WAIT_FOR_INPUT("Frg_Storage1_2_E68",TRUE)
  ;-------------------------------------------------
  ; Reset area clearence request.
  AnfStoer_Store1_2_A100=RESET_REQUEST
  ;-------------------------------------------------
  ; start cyclic clearence check
  $CYCFLAG[ciFreigabeSPS]=Frg_Storage1_2_E68
  ;-------------------------------------------------
ENDIF
;***************************************************
; set "robot in area"
RobAusStorage1_2_A68=SET_IN_AREA
;ENDFOLD
;***************************************************

;***************************************************
;FOLD Check for Teachmode
IF $FLAG[M_Teachen] THEN
  WAIT FOR $T1
ENDIF
;ENDFOLD
;***************************************************

